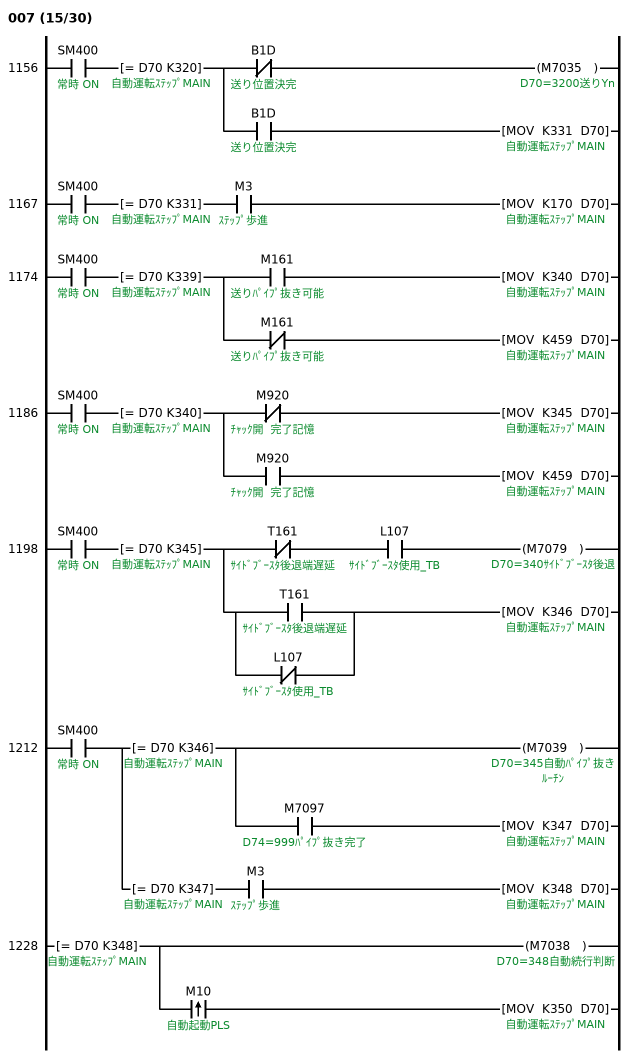
1156  LD      SM400  ; 常時 ON
      AND=    D70 K320  ; 自動運転ｽﾃｯﾌﾟMAIN
      MPS
      ANI     B1D  ; 送り位置決完
      OUT     M7035  ; D70=3200送りYn
      MPP
      AND     B1D  ; 送り位置決完
      MOV     K331 D70
1167  LD      SM400  ; 常時 ON
      AND=    D70 K331  ; 自動運転ｽﾃｯﾌﾟMAIN
      AND     M3  ; ｽﾃｯﾌﾟ歩進
      MOV     K170 D70
1174  LD      SM400  ; 常時 ON
      AND=    D70 K339  ; 自動運転ｽﾃｯﾌﾟMAIN
      MPS
      AND     M161  ; 送りﾊﾟｲﾌﾟ抜き可能
      MOV     K340 D70
      MPP
      ANI     M161  ; 送りﾊﾟｲﾌﾟ抜き可能
      MOV     K459 D70
1186  LD      SM400  ; 常時 ON
      AND=    D70 K340  ; 自動運転ｽﾃｯﾌﾟMAIN
      MPS
      ANI     M920  ; ﾁｬｯｸ開  完了記憶
      MOV     K345 D70
      MPP
      AND     M920  ; ﾁｬｯｸ開  完了記憶
      MOV     K459 D70
1198  LD      SM400  ; 常時 ON
      AND=    D70 K345  ; 自動運転ｽﾃｯﾌﾟMAIN
      MPS
      ANI     T161  ; ｻｲﾄﾞﾌﾞｰｽﾀ後退端遅延
      AND     L107  ; ｻｲﾄﾞﾌﾞｰｽﾀ使用_TB
      OUT     M7079  ; D70=340ｻｲﾄﾞﾌﾞｰｽﾀ後退
      MPP
      LD      T161  ; ｻｲﾄﾞﾌﾞｰｽﾀ後退端遅延
      ORI     L107  ; ｻｲﾄﾞﾌﾞｰｽﾀ使用_TB
      ANB
      MOV     K346 D70
1212  LD      SM400  ; 常時 ON
      MPS
      AND=    D70 K346  ; 自動運転ｽﾃｯﾌﾟMAIN
      OUT     M7039  ; D70=345自動ﾊﾟｲﾌﾟ抜きﾙｰﾁﾝ
      AND     M7097  ; D74=999ﾊﾟｲﾌﾟ抜き完了
      MOV     K347 D70
      MPP
      AND=    D70 K347  ; 自動運転ｽﾃｯﾌﾟMAIN
      AND     M3  ; ｽﾃｯﾌﾟ歩進
      MOV     K348 D70
1228  LD=     D70 K348  ; 自動運転ｽﾃｯﾌﾟMAIN
      OUT     M7038  ; D70=348自動続行判断
      ANDP    M10  ; 自動起動PLS
      MOV     K350 D70
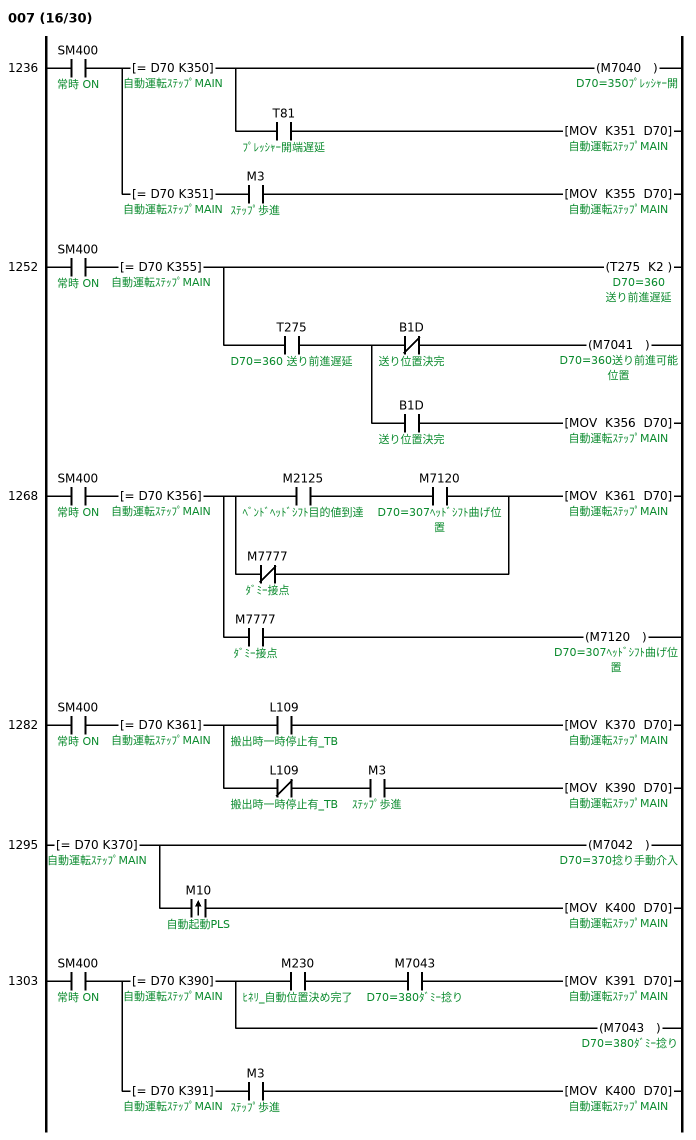
1236  LD      SM400  ; 常時 ON
      MPS
      AND=    D70 K350  ; 自動運転ｽﾃｯﾌﾟMAIN
      OUT     M7040  ; D70=350ﾌﾟﾚｯｼｬｰ開
      AND     T81  ; ﾌﾟﾚｯｼｬｰ開端遅延
      MOV     K351 D70
      MPP
      AND=    D70 K351  ; 自動運転ｽﾃｯﾌﾟMAIN
      AND     M3  ; ｽﾃｯﾌﾟ歩進
      MOV     K355 D70
1252  LD      SM400  ; 常時 ON
      AND=    D70 K355  ; 自動運転ｽﾃｯﾌﾟMAIN
      OUT     T275 K2  ; D70=360 送り前進遅延
      AND     T275  ; D70=360 送り前進遅延
      MPS
      ANI     B1D  ; 送り位置決完
      OUT     M7041  ; D70=360送り前進可能位置
      MPP
      AND     B1D  ; 送り位置決完
      MOV     K356 D70
1268  LD      SM400  ; 常時 ON
      AND=    D70 K356  ; 自動運転ｽﾃｯﾌﾟMAIN
      MPS
      LD      M2125  ; ﾍﾞﾝﾄﾞﾍｯﾄﾞｼﾌﾄ目的値到達
      AND     M7120  ; D70=307ﾍｯﾄﾞｼﾌﾄ曲げ位置
      ORI     M7777  ; ﾀﾞﾐｰ接点
      ANB
      MOV     K361 D70
      MPP
      AND     M7777  ; ﾀﾞﾐｰ接点
      OUT     M7120  ; D70=307ﾍｯﾄﾞｼﾌﾄ曲げ位置
1282  LD      SM400  ; 常時 ON
      AND=    D70 K361  ; 自動運転ｽﾃｯﾌﾟMAIN
      MPS
      AND     L109  ; 搬出時一時停止有_TB
      MOV     K370 D70
      MPP
      ANI     L109  ; 搬出時一時停止有_TB
      AND     M3  ; ｽﾃｯﾌﾟ歩進
      MOV     K390 D70
1295  LD=     D70 K370  ; 自動運転ｽﾃｯﾌﾟMAIN
      OUT     M7042  ; D70=370捻り手動介入
      ANDP    M10  ; 自動起動PLS
      MOV     K400 D70
1303  LD      SM400  ; 常時 ON
      MPS
      AND=    D70 K390  ; 自動運転ｽﾃｯﾌﾟMAIN
      MPS
      AND     M230  ; ﾋﾈﾘ_自動位置決め完了
      AND     M7043  ; D70=380ﾀﾞﾐｰ捻り
      MOV     K391 D70
      MPP
      OUT     M7043  ; D70=380ﾀﾞﾐｰ捻り
      MPP
      AND=    D70 K391  ; 自動運転ｽﾃｯﾌﾟMAIN
      AND     M3  ; ｽﾃｯﾌﾟ歩進
      MOV     K400 D70
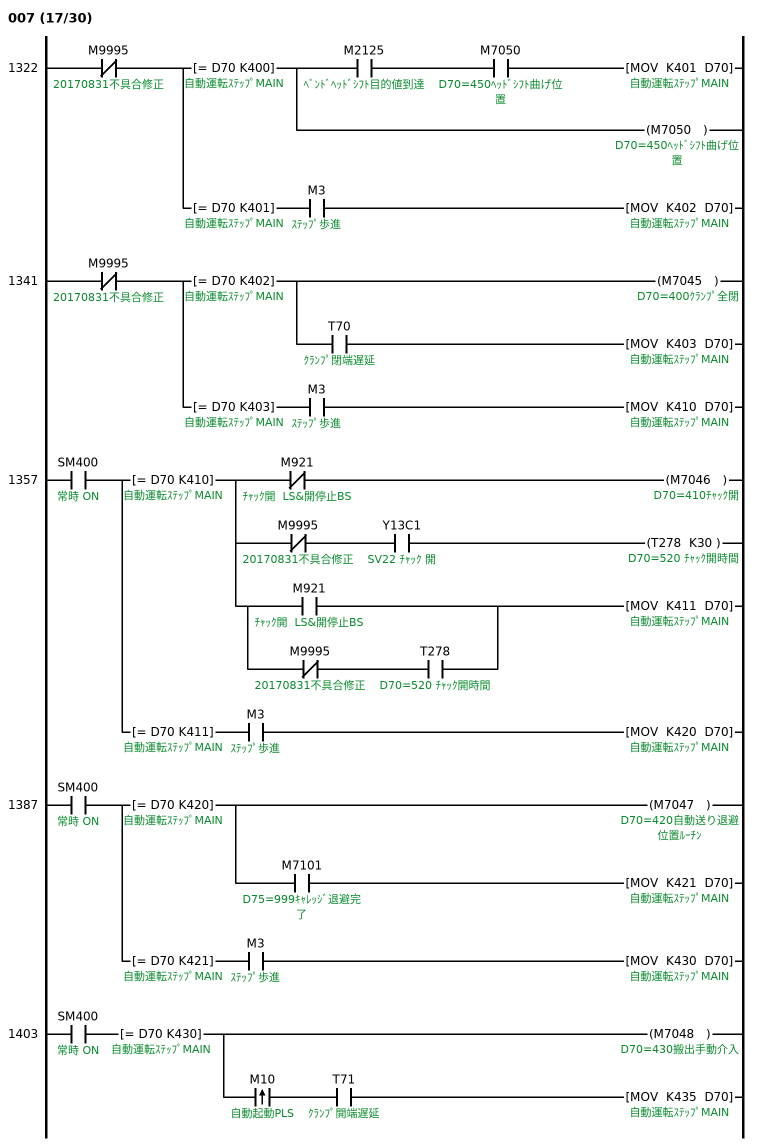
1322  LDI     M9995  ; 20170831不具合修正
      MPS
      AND=    D70 K400  ; 自動運転ｽﾃｯﾌﾟMAIN
      MPS
      AND     M2125  ; ﾍﾞﾝﾄﾞﾍｯﾄﾞｼﾌﾄ目的値到達
      AND     M7050  ; D70=450ﾍｯﾄﾞｼﾌﾄ曲げ位置
      MOV     K401 D70
      MPP
      OUT     M7050  ; D70=450ﾍｯﾄﾞｼﾌﾄ曲げ位置
      MPP
      AND=    D70 K401  ; 自動運転ｽﾃｯﾌﾟMAIN
      AND     M3  ; ｽﾃｯﾌﾟ歩進
      MOV     K402 D70
1341  LDI     M9995  ; 20170831不具合修正
      MPS
      AND=    D70 K402  ; 自動運転ｽﾃｯﾌﾟMAIN
      OUT     M7045  ; D70=400ｸﾗﾝﾌﾟ全閉
      AND     T70  ; ｸﾗﾝﾌﾟ閉端遅延
      MOV     K403 D70
      MPP
      AND=    D70 K403  ; 自動運転ｽﾃｯﾌﾟMAIN
      AND     M3  ; ｽﾃｯﾌﾟ歩進
      MOV     K410 D70
1357  LD      SM400  ; 常時 ON
      MPS
      AND=    D70 K410  ; 自動運転ｽﾃｯﾌﾟMAIN
      MPS
      ANI     M921  ; ﾁｬｯｸ開  LS&開停止BS
      OUT     M7046  ; D70=410ﾁｬｯｸ開
      MRD
      ANI     M9995  ; 20170831不具合修正
      AND     Y13C1  ; SV22 ﾁｬｯｸ 開
      OUT     T278 K30  ; D70=520 ﾁｬｯｸ開時間
      MPP
      LD      M921  ; ﾁｬｯｸ開  LS&開停止BS
      LDI     M9995  ; 20170831不具合修正
      AND     T278  ; D70=520 ﾁｬｯｸ開時間
      ORB
      ANB
      MOV     K411 D70
      MPP
      AND=    D70 K411  ; 自動運転ｽﾃｯﾌﾟMAIN
      AND     M3  ; ｽﾃｯﾌﾟ歩進
      MOV     K420 D70
1387  LD      SM400  ; 常時 ON
      MPS
      AND=    D70 K420  ; 自動運転ｽﾃｯﾌﾟMAIN
      OUT     M7047  ; D70=420自動送り退避位置ﾙｰﾁﾝ
      AND     M7101  ; D75=999ｷｬﾚｯｼﾞ退避完了
      MOV     K421 D70
      MPP
      AND=    D70 K421  ; 自動運転ｽﾃｯﾌﾟMAIN
      AND     M3  ; ｽﾃｯﾌﾟ歩進
      MOV     K430 D70
1403  LD      SM400  ; 常時 ON
      AND=    D70 K430  ; 自動運転ｽﾃｯﾌﾟMAIN
      OUT     M7048  ; D70=430搬出手動介入
      ANDP    M10  ; 自動起動PLS
      AND     T71  ; ｸﾗﾝﾌﾟ開端遅延
      MOV     K435 D70
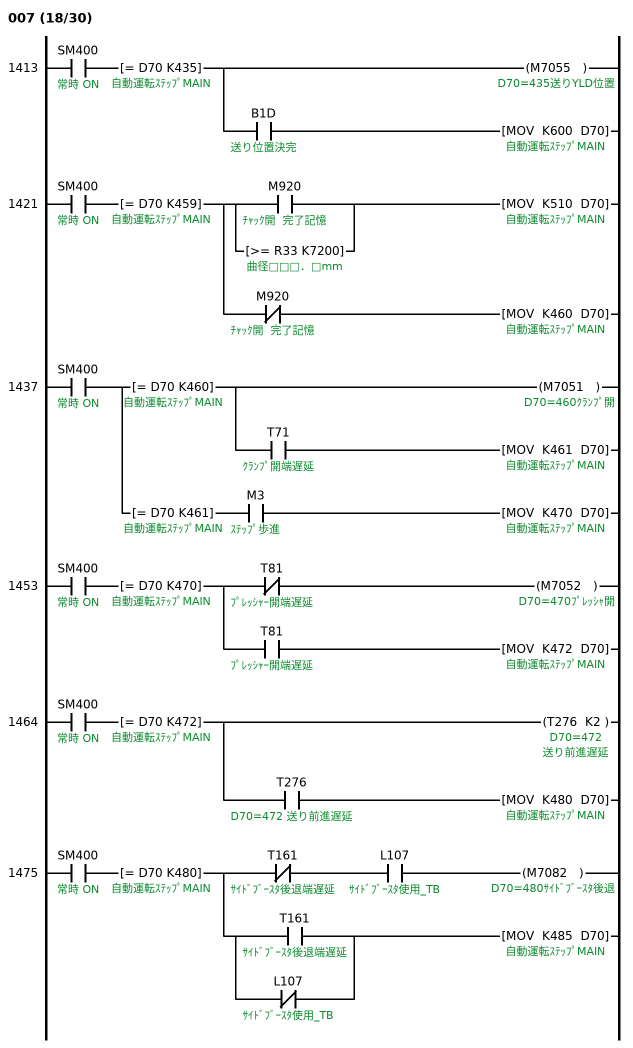
1413  LD      SM400  ; 常時 ON
      AND=    D70 K435  ; 自動運転ｽﾃｯﾌﾟMAIN
      OUT     M7055  ; D70=435送りYLD位置
      AND     B1D  ; 送り位置決完
      MOV     K600 D70
1421  LD      SM400  ; 常時 ON
      AND=    D70 K459  ; 自動運転ｽﾃｯﾌﾟMAIN
      MPS
      LD      M920  ; ﾁｬｯｸ開  完了記憶
      OR>=    R33 K7200  ; 曲径□□□．□mm
      ANB
      MOV     K510 D70
      MPP
      ANI     M920  ; ﾁｬｯｸ開  完了記憶
      MOV     K460 D70
1437  LD      SM400  ; 常時 ON
      MPS
      AND=    D70 K460  ; 自動運転ｽﾃｯﾌﾟMAIN
      OUT     M7051  ; D70=460ｸﾗﾝﾌﾟ開
      AND     T71  ; ｸﾗﾝﾌﾟ開端遅延
      MOV     K461 D70
      MPP
      AND=    D70 K461  ; 自動運転ｽﾃｯﾌﾟMAIN
      AND     M3  ; ｽﾃｯﾌﾟ歩進
      MOV     K470 D70
1453  LD      SM400  ; 常時 ON
      AND=    D70 K470  ; 自動運転ｽﾃｯﾌﾟMAIN
      MPS
      ANI     T81  ; ﾌﾟﾚｯｼｬｰ開端遅延
      OUT     M7052  ; D70=470ﾌﾟﾚｯｼｬ開
      MPP
      AND     T81  ; ﾌﾟﾚｯｼｬｰ開端遅延
      MOV     K472 D70
1464  LD      SM400  ; 常時 ON
      AND=    D70 K472  ; 自動運転ｽﾃｯﾌﾟMAIN
      OUT     T276 K2  ; D70=472 送り前進遅延
      AND     T276  ; D70=472 送り前進遅延
      MOV     K480 D70
1475  LD      SM400  ; 常時 ON
      AND=    D70 K480  ; 自動運転ｽﾃｯﾌﾟMAIN
      MPS
      ANI     T161  ; ｻｲﾄﾞﾌﾞｰｽﾀ後退端遅延
      AND     L107  ; ｻｲﾄﾞﾌﾞｰｽﾀ使用_TB
      OUT     M7082  ; D70=480ｻｲﾄﾞﾌﾞｰｽﾀ後退
      MPP
      LD      T161  ; ｻｲﾄﾞﾌﾞｰｽﾀ後退端遅延
      ORI     L107  ; ｻｲﾄﾞﾌﾞｰｽﾀ使用_TB
      ANB
      MOV     K485 D70
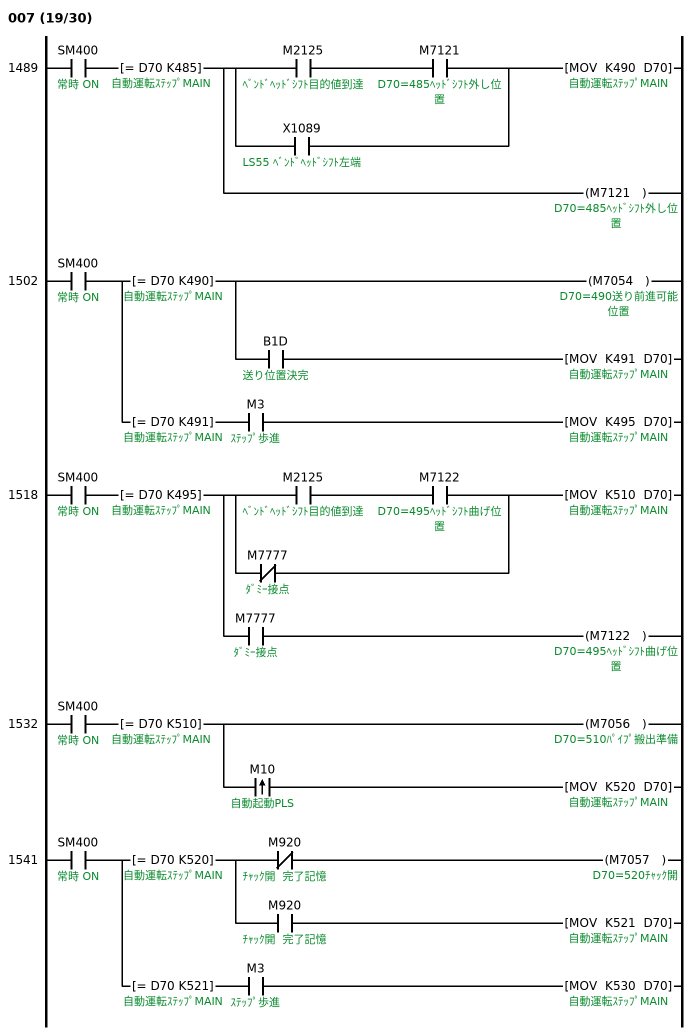
1489  LD      SM400  ; 常時 ON
      AND=    D70 K485  ; 自動運転ｽﾃｯﾌﾟMAIN
      MPS
      LD      M2125  ; ﾍﾞﾝﾄﾞﾍｯﾄﾞｼﾌﾄ目的値到達
      AND     M7121  ; D70=485ﾍｯﾄﾞｼﾌﾄ外し位置
      OR      X1089  ; LS55 ﾍﾞﾝﾄﾞﾍｯﾄﾞｼﾌﾄ左端
      ANB
      MOV     K490 D70
      MPP
      OUT     M7121  ; D70=485ﾍｯﾄﾞｼﾌﾄ外し位置
1502  LD      SM400  ; 常時 ON
      MPS
      AND=    D70 K490  ; 自動運転ｽﾃｯﾌﾟMAIN
      OUT     M7054  ; D70=490送り前進可能位置
      AND     B1D  ; 送り位置決完
      MOV     K491 D70
      MPP
      AND=    D70 K491  ; 自動運転ｽﾃｯﾌﾟMAIN
      AND     M3  ; ｽﾃｯﾌﾟ歩進
      MOV     K495 D70
1518  LD      SM400  ; 常時 ON
      AND=    D70 K495  ; 自動運転ｽﾃｯﾌﾟMAIN
      MPS
      LD      M2125  ; ﾍﾞﾝﾄﾞﾍｯﾄﾞｼﾌﾄ目的値到達
      AND     M7122  ; D70=495ﾍｯﾄﾞｼﾌﾄ曲げ位置
      ORI     M7777  ; ﾀﾞﾐｰ接点
      ANB
      MOV     K510 D70
      MPP
      AND     M7777  ; ﾀﾞﾐｰ接点
      OUT     M7122  ; D70=495ﾍｯﾄﾞｼﾌﾄ曲げ位置
1532  LD      SM400  ; 常時 ON
      AND=    D70 K510  ; 自動運転ｽﾃｯﾌﾟMAIN
      OUT     M7056  ; D70=510ﾊﾟｲﾌﾟ搬出準備
      ANDP    M10  ; 自動起動PLS
      MOV     K520 D70
1541  LD      SM400  ; 常時 ON
      MPS
      AND=    D70 K520  ; 自動運転ｽﾃｯﾌﾟMAIN
      MPS
      ANI     M920  ; ﾁｬｯｸ開  完了記憶
      OUT     M7057  ; D70=520ﾁｬｯｸ開
      MPP
      AND     M920  ; ﾁｬｯｸ開  完了記憶
      MOV     K521 D70
      MPP
      AND=    D70 K521  ; 自動運転ｽﾃｯﾌﾟMAIN
      AND     M3  ; ｽﾃｯﾌﾟ歩進
      MOV     K530 D70
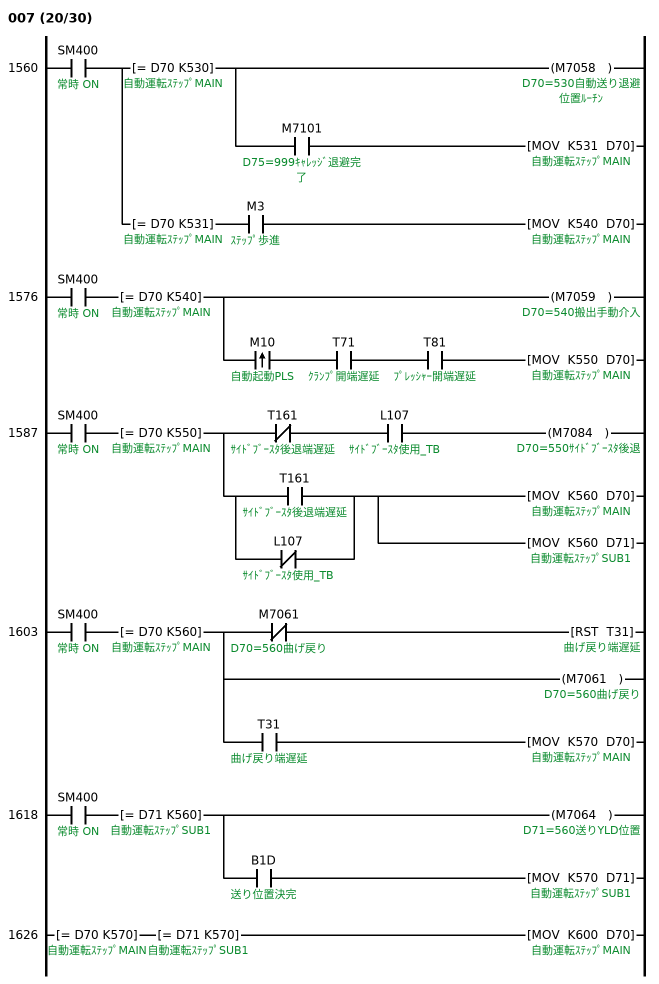
1560  LD      SM400  ; 常時 ON
      MPS
      AND=    D70 K530  ; 自動運転ｽﾃｯﾌﾟMAIN
      OUT     M7058  ; D70=530自動送り退避位置ﾙｰﾁﾝ
      AND     M7101  ; D75=999ｷｬﾚｯｼﾞ退避完了
      MOV     K531 D70
      MPP
      AND=    D70 K531  ; 自動運転ｽﾃｯﾌﾟMAIN
      AND     M3  ; ｽﾃｯﾌﾟ歩進
      MOV     K540 D70
1576  LD      SM400  ; 常時 ON
      AND=    D70 K540  ; 自動運転ｽﾃｯﾌﾟMAIN
      OUT     M7059  ; D70=540搬出手動介入
      ANDP    M10  ; 自動起動PLS
      AND     T71  ; ｸﾗﾝﾌﾟ開端遅延
      AND     T81  ; ﾌﾟﾚｯｼｬｰ開端遅延
      MOV     K550 D70
1587  LD      SM400  ; 常時 ON
      AND=    D70 K550  ; 自動運転ｽﾃｯﾌﾟMAIN
      MPS
      ANI     T161  ; ｻｲﾄﾞﾌﾞｰｽﾀ後退端遅延
      AND     L107  ; ｻｲﾄﾞﾌﾞｰｽﾀ使用_TB
      OUT     M7084  ; D70=550ｻｲﾄﾞﾌﾞｰｽﾀ後退
      MPP
      LD      T161  ; ｻｲﾄﾞﾌﾞｰｽﾀ後退端遅延
      ORI     L107  ; ｻｲﾄﾞﾌﾞｰｽﾀ使用_TB
      ANB
      MOV     K560 D70
      MOV     K560 D71
1603  LD      SM400  ; 常時 ON
      AND=    D70 K560  ; 自動運転ｽﾃｯﾌﾟMAIN
      MPS
      ANI     M7061  ; D70=560曲げ戻り
      RST     T31  ; 曲げ戻り端遅延
      MPP
      OUT     M7061  ; D70=560曲げ戻り
      AND     T31  ; 曲げ戻り端遅延
      MOV     K570 D70
1618  LD      SM400  ; 常時 ON
      AND=    D71 K560  ; 自動運転ｽﾃｯﾌﾟSUB1
      OUT     M7064  ; D71=560送りYLD位置
      AND     B1D  ; 送り位置決完
      MOV     K570 D71
1626  LD=     D70 K570  ; 自動運転ｽﾃｯﾌﾟMAIN
      AND=    D71 K570  ; 自動運転ｽﾃｯﾌﾟSUB1
      MOV     K600 D70
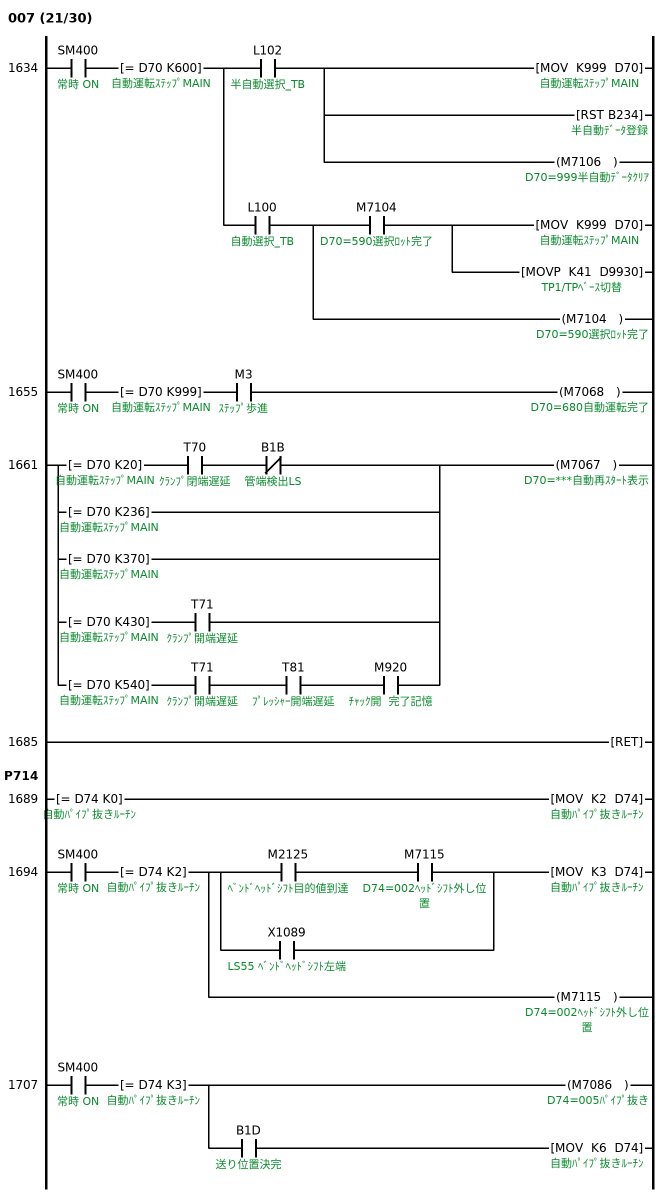
1634  LD      SM400  ; 常時 ON
      AND=    D70 K600  ; 自動運転ｽﾃｯﾌﾟMAIN
      MPS
      AND     L102  ; 半自動選択_TB
      MOV     K999 D70
      RST     B234  ; 半自動ﾃﾞｰﾀ登録
      OUT     M7106  ; D70=999半自動ﾃﾞｰﾀｸﾘｱ
      MPP
      AND     L100  ; 自動選択_TB
      MPS
      AND     M7104  ; D70=590選択ﾛｯﾄ完了
      MOV     K999 D70
      MOVP    K41 D9930  ; TP1/TPﾍﾞｰｽ切替
      MPP
      OUT     M7104  ; D70=590選択ﾛｯﾄ完了
1655  LD      SM400  ; 常時 ON
      AND=    D70 K999  ; 自動運転ｽﾃｯﾌﾟMAIN
      AND     M3  ; ｽﾃｯﾌﾟ歩進
      OUT     M7068  ; D70=680自動運転完了
1661  LD=     D70 K20  ; 自動運転ｽﾃｯﾌﾟMAIN
      AND     T70  ; ｸﾗﾝﾌﾟ閉端遅延
      ANI     B1B  ; 管端検出LS
      OR=     D70 K236  ; 自動運転ｽﾃｯﾌﾟMAIN
      OR=     D70 K370  ; 自動運転ｽﾃｯﾌﾟMAIN
      LD=     D70 K430  ; 自動運転ｽﾃｯﾌﾟMAIN
      AND     T71  ; ｸﾗﾝﾌﾟ開端遅延
      ORB
      LD=     D70 K540  ; 自動運転ｽﾃｯﾌﾟMAIN
      AND     T71  ; ｸﾗﾝﾌﾟ開端遅延
      AND     T81  ; ﾌﾟﾚｯｼｬｰ開端遅延
      AND     M920  ; ﾁｬｯｸ開  完了記憶
      ORB
      OUT     M7067  ; D70=***自動再ｽﾀｰﾄ表示
1685  RET
; 
      P714
1689  LD=     D74 K0  ; 自動ﾊﾟｲﾌﾟ抜きﾙｰﾁﾝ
      MOV     K2 D74
1694  LD      SM400  ; 常時 ON
      AND=    D74 K2  ; 自動ﾊﾟｲﾌﾟ抜きﾙｰﾁﾝ
      MPS
      LD      M2125  ; ﾍﾞﾝﾄﾞﾍｯﾄﾞｼﾌﾄ目的値到達
      AND     M7115  ; D74=002ﾍｯﾄﾞｼﾌﾄ外し位置
      OR      X1089  ; LS55 ﾍﾞﾝﾄﾞﾍｯﾄﾞｼﾌﾄ左端
      ANB
      MOV     K3 D74
      MPP
      OUT     M7115  ; D74=002ﾍｯﾄﾞｼﾌﾄ外し位置
1707  LD      SM400  ; 常時 ON
      AND=    D74 K3  ; 自動ﾊﾟｲﾌﾟ抜きﾙｰﾁﾝ
      OUT     M7086  ; D74=005ﾊﾟｲﾌﾟ抜き
      AND     B1D  ; 送り位置決完
      MOV     K6 D74
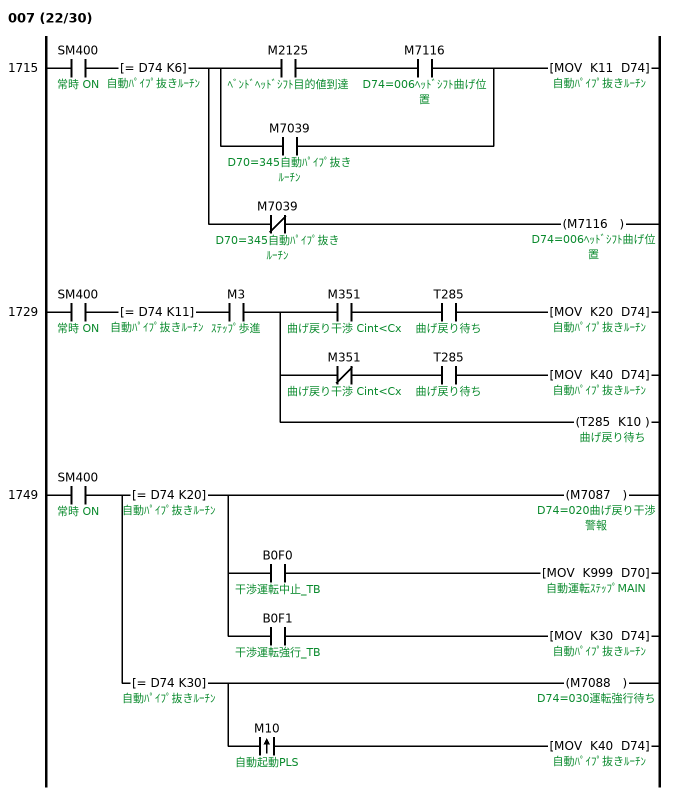
1715  LD      SM400  ; 常時 ON
      AND=    D74 K6  ; 自動ﾊﾟｲﾌﾟ抜きﾙｰﾁﾝ
      MPS
      LD      M2125  ; ﾍﾞﾝﾄﾞﾍｯﾄﾞｼﾌﾄ目的値到達
      AND     M7116  ; D74=006ﾍｯﾄﾞｼﾌﾄ曲げ位置
      OR      M7039  ; D70=345自動ﾊﾟｲﾌﾟ抜きﾙｰﾁﾝ
      ANB
      MOV     K11 D74
      MPP
      ANI     M7039  ; D70=345自動ﾊﾟｲﾌﾟ抜きﾙｰﾁﾝ
      OUT     M7116  ; D74=006ﾍｯﾄﾞｼﾌﾄ曲げ位置
1729  LD      SM400  ; 常時 ON
      AND=    D74 K11  ; 自動ﾊﾟｲﾌﾟ抜きﾙｰﾁﾝ
      AND     M3  ; ｽﾃｯﾌﾟ歩進
      MPS
      AND     M351  ; 曲げ戻り干渉 Cint<Cx
      AND     T285  ; 曲げ戻り待ち
      MOV     K20 D74
      MRD
      ANI     M351  ; 曲げ戻り干渉 Cint<Cx
      AND     T285  ; 曲げ戻り待ち
      MOV     K40 D74
      MPP
      OUT     T285 K10  ; 曲げ戻り待ち
1749  LD      SM400  ; 常時 ON
      MPS
      AND=    D74 K20  ; 自動ﾊﾟｲﾌﾟ抜きﾙｰﾁﾝ
      OUT     M7087  ; D74=020曲げ戻り干渉警報
      MPS
      AND     B0F0  ; 干渉運転中止_TB
      MOV     K999 D70
      MPP
      AND     B0F1  ; 干渉運転強行_TB
      MOV     K30 D74
      MPP
      AND=    D74 K30  ; 自動ﾊﾟｲﾌﾟ抜きﾙｰﾁﾝ
      OUT     M7088  ; D74=030運転強行待ち
      ANDP    M10  ; 自動起動PLS
      MOV     K40 D74
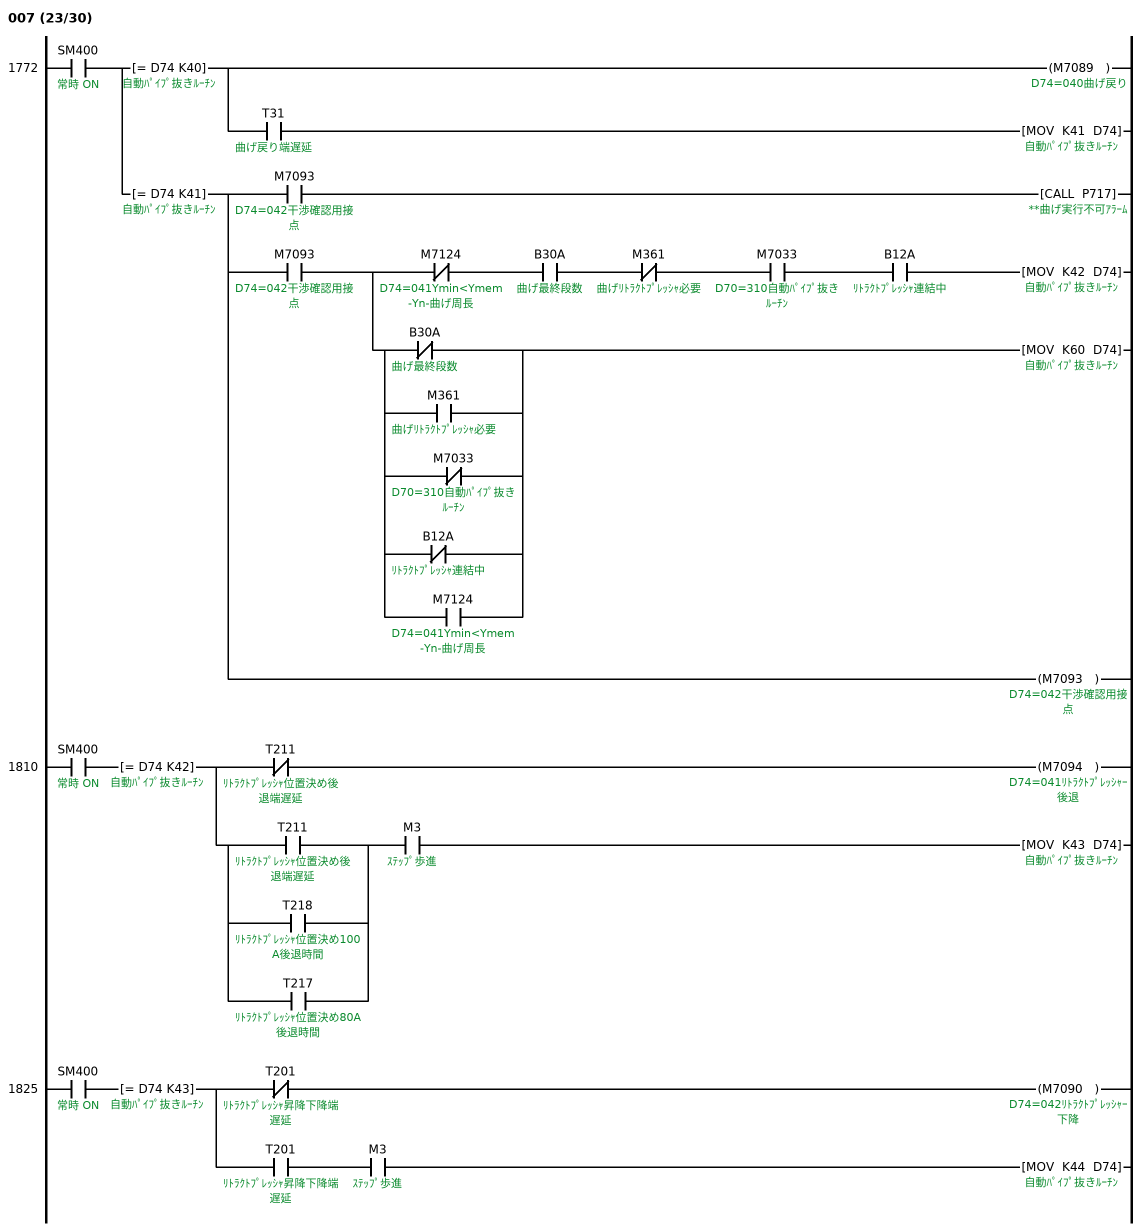
1772  LD      SM400  ; 常時 ON
      MPS
      AND=    D74 K40  ; 自動ﾊﾟｲﾌﾟ抜きﾙｰﾁﾝ
      OUT     M7089  ; D74=040曲げ戻り
      AND     T31  ; 曲げ戻り端遅延
      MOV     K41 D74
      MPP
      AND=    D74 K41  ; 自動ﾊﾟｲﾌﾟ抜きﾙｰﾁﾝ
      MPS
      AND     M7093  ; D74=042干渉確認用接点
      CALL    P717
      MRD
      AND     M7093  ; D74=042干渉確認用接点
      MPS
      ANI     M7124  ; D74=041Ymin<Ymem-Yn-曲げ周長
      AND     B30A  ; 曲げ最終段数
      ANI     M361  ; 曲げﾘﾄﾗｸﾄﾌﾟﾚｯｼｬ必要
      AND     M7033  ; D70=310自動ﾊﾟｲﾌﾟ抜きﾙｰﾁﾝ
      AND     B12A  ; ﾘﾄﾗｸﾄﾌﾟﾚｯｼｬ連結中
      MOV     K42 D74
      MPP
      LDI     B30A  ; 曲げ最終段数
      OR      M361  ; 曲げﾘﾄﾗｸﾄﾌﾟﾚｯｼｬ必要
      ORI     M7033  ; D70=310自動ﾊﾟｲﾌﾟ抜きﾙｰﾁﾝ
      ORI     B12A  ; ﾘﾄﾗｸﾄﾌﾟﾚｯｼｬ連結中
      OR      M7124  ; D74=041Ymin<Ymem-Yn-曲げ周長
      ANB
      MOV     K60 D74
      MPP
      OUT     M7093  ; D74=042干渉確認用接点
1810  LD      SM400  ; 常時 ON
      AND=    D74 K42  ; 自動ﾊﾟｲﾌﾟ抜きﾙｰﾁﾝ
      MPS
      ANI     T211  ; ﾘﾄﾗｸﾄﾌﾟﾚｯｼｬ位置決め後退端遅延
      OUT     M7094  ; D74=041ﾘﾄﾗｸﾄﾌﾟﾚｯｼｬｰ後退
      MPP
      LD      T211  ; ﾘﾄﾗｸﾄﾌﾟﾚｯｼｬ位置決め後退端遅延
      OR      T218  ; ﾘﾄﾗｸﾄﾌﾟﾚｯｼｬ位置決め100A後退時間
      OR      T217  ; ﾘﾄﾗｸﾄﾌﾟﾚｯｼｬ位置決め80A後退時間
      ANB
      AND     M3  ; ｽﾃｯﾌﾟ歩進
      MOV     K43 D74
1825  LD      SM400  ; 常時 ON
      AND=    D74 K43  ; 自動ﾊﾟｲﾌﾟ抜きﾙｰﾁﾝ
      MPS
      ANI     T201  ; ﾘﾄﾗｸﾄﾌﾟﾚｯｼｬ昇降下降端遅延
      OUT     M7090  ; D74=042ﾘﾄﾗｸﾄﾌﾟﾚｯｼｬｰ下降
      MPP
      AND     T201  ; ﾘﾄﾗｸﾄﾌﾟﾚｯｼｬ昇降下降端遅延
      AND     M3  ; ｽﾃｯﾌﾟ歩進
      MOV     K44 D74
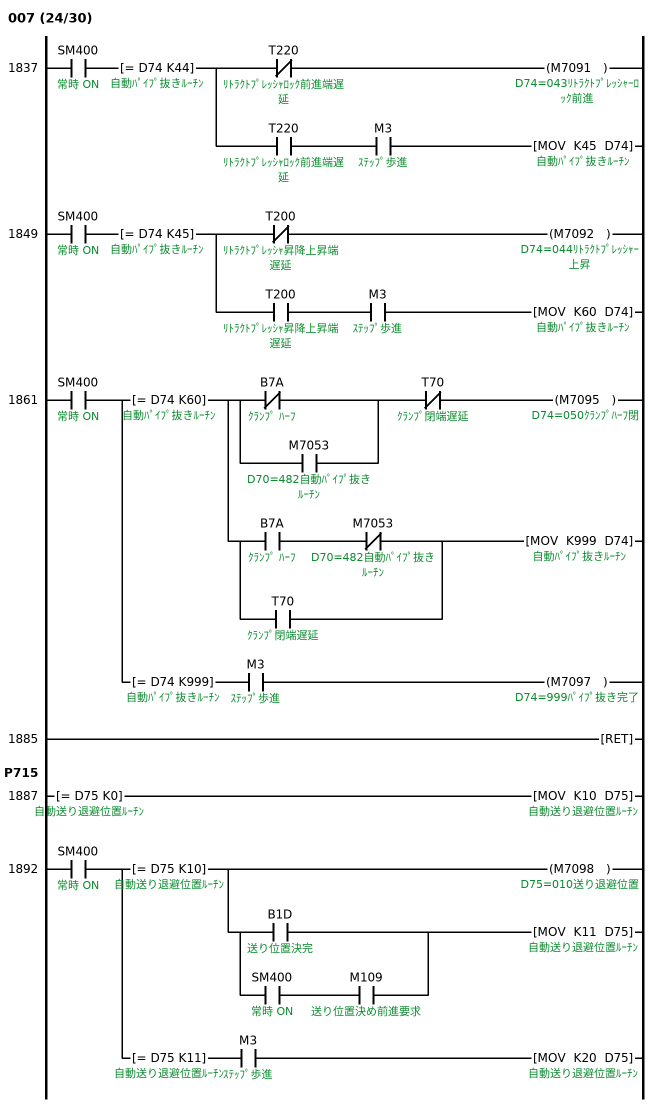
1837  LD      SM400  ; 常時 ON
      AND=    D74 K44  ; 自動ﾊﾟｲﾌﾟ抜きﾙｰﾁﾝ
      MPS
      ANI     T220  ; ﾘﾄﾗｸﾄﾌﾟﾚｯｼｬﾛｯｸ前進端遅延
      OUT     M7091  ; D74=043ﾘﾄﾗｸﾄﾌﾟﾚｯｼｬｰﾛｯｸ前進
      MPP
      AND     T220  ; ﾘﾄﾗｸﾄﾌﾟﾚｯｼｬﾛｯｸ前進端遅延
      AND     M3  ; ｽﾃｯﾌﾟ歩進
      MOV     K45 D74
1849  LD      SM400  ; 常時 ON
      AND=    D74 K45  ; 自動ﾊﾟｲﾌﾟ抜きﾙｰﾁﾝ
      MPS
      ANI     T200  ; ﾘﾄﾗｸﾄﾌﾟﾚｯｼｬ昇降上昇端遅延
      OUT     M7092  ; D74=044ﾘﾄﾗｸﾄﾌﾟﾚｯｼｬｰ上昇
      MPP
      AND     T200  ; ﾘﾄﾗｸﾄﾌﾟﾚｯｼｬ昇降上昇端遅延
      AND     M3  ; ｽﾃｯﾌﾟ歩進
      MOV     K60 D74
1861  LD      SM400  ; 常時 ON
      MPS
      AND=    D74 K60  ; 自動ﾊﾟｲﾌﾟ抜きﾙｰﾁﾝ
      MPS
      LDI     B7A  ; ｸﾗﾝﾌﾟ ﾊｰﾌ
      OR      M7053  ; D70=482自動ﾊﾟｲﾌﾟ抜きﾙｰﾁﾝ
      ANB
      ANI     T70  ; ｸﾗﾝﾌﾟ閉端遅延
      OUT     M7095  ; D74=050ｸﾗﾝﾌﾟﾊｰﾌ閉
      MPP
      LD      B7A  ; ｸﾗﾝﾌﾟ ﾊｰﾌ
      ANI     M7053  ; D70=482自動ﾊﾟｲﾌﾟ抜きﾙｰﾁﾝ
      OR      T70  ; ｸﾗﾝﾌﾟ閉端遅延
      ANB
      MOV     K999 D74
      MPP
      AND=    D74 K999  ; 自動ﾊﾟｲﾌﾟ抜きﾙｰﾁﾝ
      AND     M3  ; ｽﾃｯﾌﾟ歩進
      OUT     M7097  ; D74=999ﾊﾟｲﾌﾟ抜き完了
1885  RET
      P715
1887  LD=     D75 K0  ; 自動送り退避位置ﾙｰﾁﾝ
      MOV     K10 D75
1892  LD      SM400  ; 常時 ON
      MPS
      AND=    D75 K10  ; 自動送り退避位置ﾙｰﾁﾝ
      OUT     M7098  ; D75=010送り退避位置
      LD      B1D  ; 送り位置決完
      LD      SM400  ; 常時 ON
      AND     M109  ; 送り位置決め前進要求
      ORB
      ANB
      MOV     K11 D75
      MPP
      AND=    D75 K11  ; 自動送り退避位置ﾙｰﾁﾝ
      AND     M3  ; ｽﾃｯﾌﾟ歩進
      MOV     K20 D75
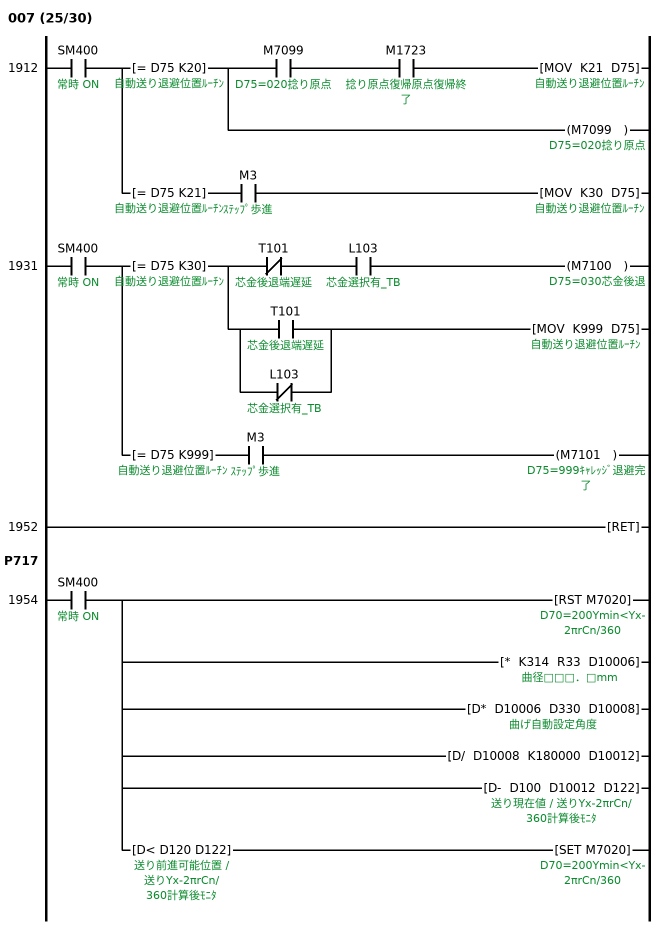
1912  LD      SM400  ; 常時 ON
      MPS
      AND=    D75 K20  ; 自動送り退避位置ﾙｰﾁﾝ
      MPS
      AND     M7099  ; D75=020捻り原点
      AND     M1723  ; 捻り原点復帰原点復帰終了
      MOV     K21 D75
      MPP
      OUT     M7099  ; D75=020捻り原点
      MPP
      AND=    D75 K21  ; 自動送り退避位置ﾙｰﾁﾝ
      AND     M3  ; ｽﾃｯﾌﾟ歩進
      MOV     K30 D75
1931  LD      SM400  ; 常時 ON
      MPS
      AND=    D75 K30  ; 自動送り退避位置ﾙｰﾁﾝ
      MPS
      ANI     T101  ; 芯金後退端遅延
      AND     L103  ; 芯金選択有_TB
      OUT     M7100  ; D75=030芯金後退
      MPP
      LD      T101  ; 芯金後退端遅延
      ORI     L103  ; 芯金選択有_TB
      ANB
      MOV     K999 D75
      MPP
      AND=    D75 K999  ; 自動送り退避位置ﾙｰﾁﾝ
      AND     M3  ; ｽﾃｯﾌﾟ歩進
      OUT     M7101  ; D75=999ｷｬﾚｯｼﾞ退避完了
1952  RET
      P717
1954  LD      SM400  ; 常時 ON
      RST     M7020  ; D70=200Ymin<Yx-2πrCn/360
      *       K314 R33 D10006
      D*      D10006 D330 D10008  ; 曲げ自動設定角度
      D/      D10008 K180000 D10012
      D-      D100 D10012 D122  ; 送りYx-2πrCn/360計算後ﾓﾆﾀ
      ANDD<   D120 D122  ; 送り前進可能位置 / 送りYx-2πrCn/360計算後ﾓﾆﾀ
      SET     M7020  ; D70=200Ymin<Yx-2πrCn/360
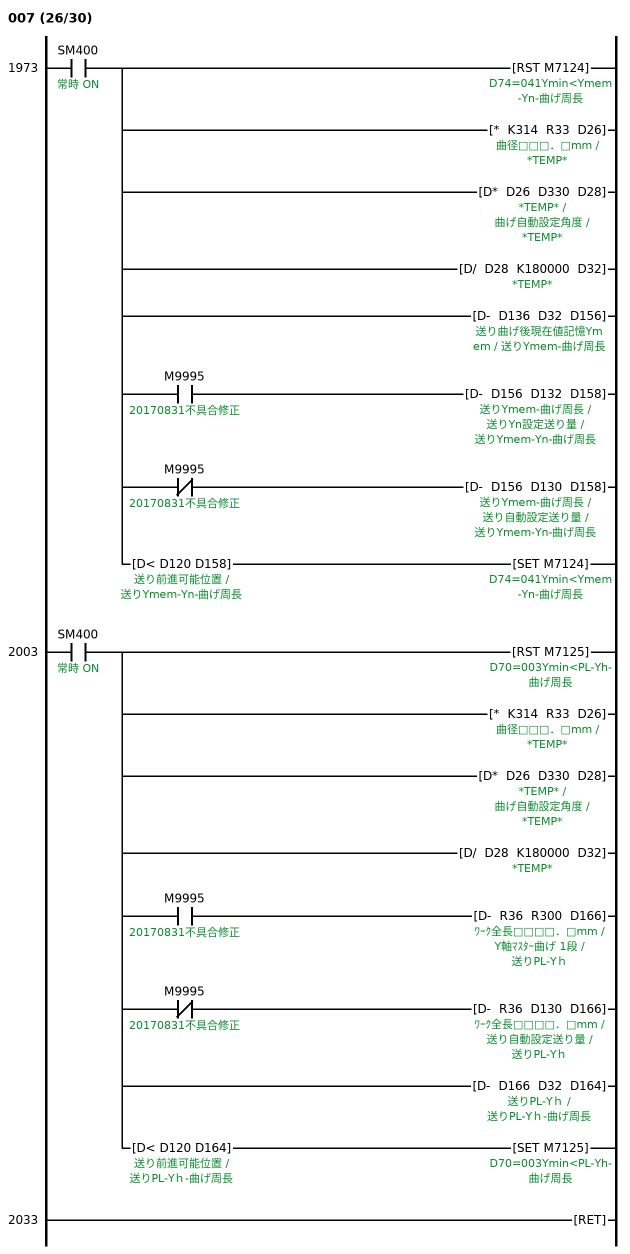
1973  LD      SM400  ; 常時 ON
      RST     M7124  ; D74=041Ymin<Ymem-Yn-曲げ周長
      *       K314 R33 D26  ; *TEMP*
      D*      D26 D330 D28  ; *TEMP*
      D/      D28 K180000 D32
      D-      D136 D32 D156  ; 送りYmem-曲げ周長
      MPS
      AND     M9995  ; 20170831不具合修正
      D-      D156 D132 D158  ; 送りYn設定送り量 / 送りYmem-Yn-曲げ周長
      MRD
      ANI     M9995  ; 20170831不具合修正
      D-      D156 D130 D158  ; 送り自動設定送り量
      MPP
      ANDD<   D120 D158  ; 送り前進可能位置 / 送りYmem-Yn-曲げ周長
      SET     M7124  ; D74=041Ymin<Ymem-Yn-曲げ周長
2003  LD      SM400  ; 常時 ON
      RST     M7125  ; D70=003Ymin<PL-Yh-曲げ周長
      *       K314 R33 D26
      D*      D26 D330 D28
      D/      D28 K180000 D32
      MPS
      AND     M9995  ; 20170831不具合修正
      D-      R36 R300 D166  ; ﾜｰｸ全長□□□□．□mm / Y軸ﾏｽﾀｰ曲げ 1段 / 送りPL-Yｈ
      MRD
      ANI     M9995  ; 20170831不具合修正
      D-      R36 D130 D166
      MPP
      D-      D166 D32 D164  ; 送りPL-Yｈ-曲げ周長
      ANDD<   D120 D164  ; 送り前進可能位置 / 送りPL-Yｈ-曲げ周長
      SET     M7125  ; D70=003Ymin<PL-Yh-曲げ周長
2033  RET
; 
      P720
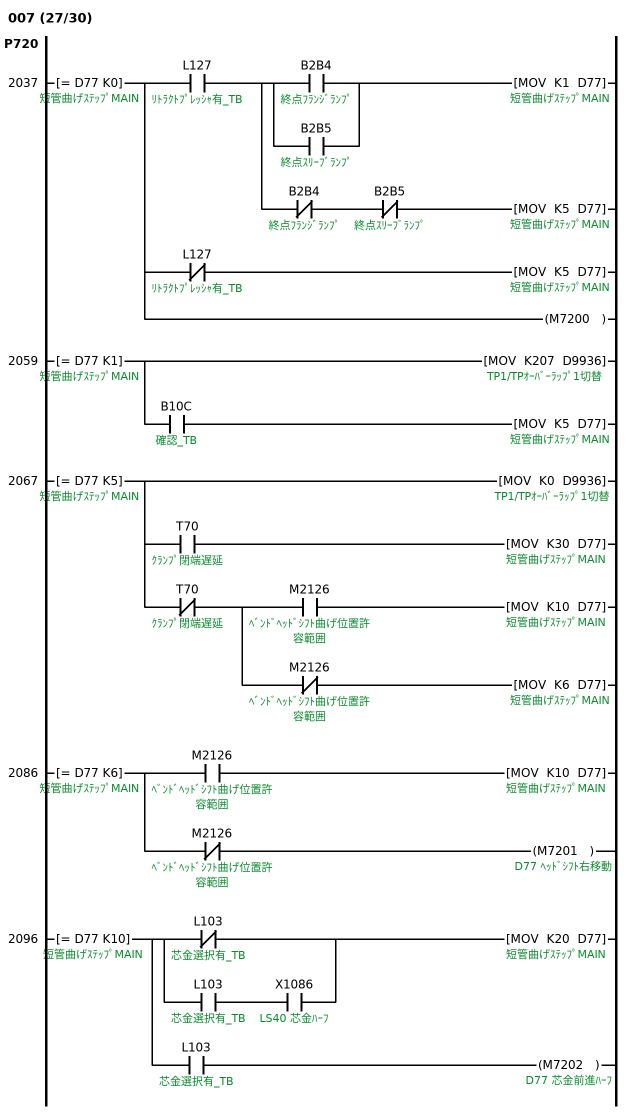
2037  LD=     D77 K0  ; 短管曲げｽﾃｯﾌﾟMAIN
      MPS
      AND     L127  ; ﾘﾄﾗｸﾄﾌﾟﾚｯｼｬ有_TB
      MPS
      LD      B2B4  ; 終点ﾌﾗﾝｼﾞﾗﾝﾌﾟ
      OR      B2B5  ; 終点ｽﾘｰﾌﾞﾗﾝﾌﾟ
      ANB
      MOV     K1 D77
      MPP
      ANI     B2B4  ; 終点ﾌﾗﾝｼﾞﾗﾝﾌﾟ
      ANI     B2B5  ; 終点ｽﾘｰﾌﾞﾗﾝﾌﾟ
      MOV     K5 D77
      MRD
      ANI     L127  ; ﾘﾄﾗｸﾄﾌﾟﾚｯｼｬ有_TB
      MOV     K5 D77
      MPP
      OUT     M7200
2059  LD=     D77 K1  ; 短管曲げｽﾃｯﾌﾟMAIN
      MOV     K207 D9936
      AND     B10C  ; 確認_TB
      MOV     K5 D77
2067  LD=     D77 K5  ; 短管曲げｽﾃｯﾌﾟMAIN
      MOV     K0 D9936
      MPS
      AND     T70  ; ｸﾗﾝﾌﾟ閉端遅延
      MOV     K30 D77
      MPP
      ANI     T70  ; ｸﾗﾝﾌﾟ閉端遅延
      MPS
      AND     M2126  ; ﾍﾞﾝﾄﾞﾍｯﾄﾞｼﾌﾄ曲げ位置許容範囲
      MOV     K10 D77
      MPP
      ANI     M2126  ; ﾍﾞﾝﾄﾞﾍｯﾄﾞｼﾌﾄ曲げ位置許容範囲
      MOV     K6 D77
2086  LD=     D77 K6  ; 短管曲げｽﾃｯﾌﾟMAIN
      MPS
      AND     M2126  ; ﾍﾞﾝﾄﾞﾍｯﾄﾞｼﾌﾄ曲げ位置許容範囲
      MOV     K10 D77
      MPP
      ANI     M2126  ; ﾍﾞﾝﾄﾞﾍｯﾄﾞｼﾌﾄ曲げ位置許容範囲
      OUT     M7201  ; D77 ﾍｯﾄﾞｼﾌﾄ右移動
2096  LD=     D77 K10  ; 短管曲げｽﾃｯﾌﾟMAIN
      MPS
      LDI     L103  ; 芯金選択有_TB
      LD      L103  ; 芯金選択有_TB
      AND     X1086  ; LS40 芯金ﾊｰﾌ
      ORB
      ANB
      MOV     K20 D77
      MPP
      AND     L103  ; 芯金選択有_TB
      OUT     M7202  ; D77 芯金前進ﾊｰﾌ
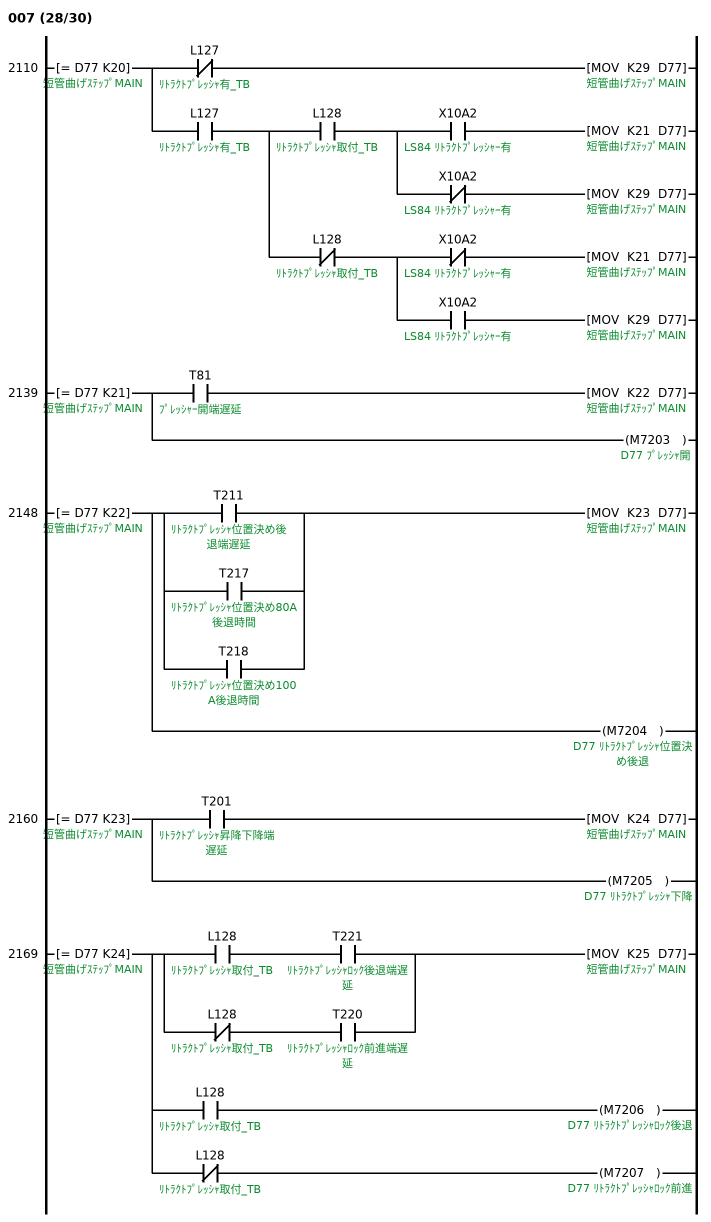
2110  LD=     D77 K20  ; 短管曲げｽﾃｯﾌﾟMAIN
      MPS
      ANI     L127  ; ﾘﾄﾗｸﾄﾌﾟﾚｯｼｬ有_TB
      MOV     K29 D77
      MPP
      AND     L127  ; ﾘﾄﾗｸﾄﾌﾟﾚｯｼｬ有_TB
      MPS
      AND     L128  ; ﾘﾄﾗｸﾄﾌﾟﾚｯｼｬ取付_TB
      MPS
      AND     X10A2  ; LS84 ﾘﾄﾗｸﾄﾌﾟﾚｯｼｬｰ有
      MOV     K21 D77
      MPP
      ANI     X10A2  ; LS84 ﾘﾄﾗｸﾄﾌﾟﾚｯｼｬｰ有
      MOV     K29 D77
      MPP
      ANI     L128  ; ﾘﾄﾗｸﾄﾌﾟﾚｯｼｬ取付_TB
      MPS
      ANI     X10A2  ; LS84 ﾘﾄﾗｸﾄﾌﾟﾚｯｼｬｰ有
      MOV     K21 D77
      MPP
      AND     X10A2  ; LS84 ﾘﾄﾗｸﾄﾌﾟﾚｯｼｬｰ有
      MOV     K29 D77
2139  LD=     D77 K21  ; 短管曲げｽﾃｯﾌﾟMAIN
      MPS
      AND     T81  ; ﾌﾟﾚｯｼｬｰ開端遅延
      MOV     K22 D77
      MPP
      OUT     M7203  ; D77 ﾌﾟﾚｯｼｬ開
2148  LD=     D77 K22  ; 短管曲げｽﾃｯﾌﾟMAIN
      MPS
      LD      T211  ; ﾘﾄﾗｸﾄﾌﾟﾚｯｼｬ位置決め後退端遅延
      OR      T217  ; ﾘﾄﾗｸﾄﾌﾟﾚｯｼｬ位置決め80A後退時間
      OR      T218  ; ﾘﾄﾗｸﾄﾌﾟﾚｯｼｬ位置決め100A後退時間
      ANB
      MOV     K23 D77
      MPP
      OUT     M7204  ; D77 ﾘﾄﾗｸﾄﾌﾟﾚｯｼｬ位置決め後退
2160  LD=     D77 K23  ; 短管曲げｽﾃｯﾌﾟMAIN
      MPS
      AND     T201  ; ﾘﾄﾗｸﾄﾌﾟﾚｯｼｬ昇降下降端遅延
      MOV     K24 D77
      MPP
      OUT     M7205  ; D77 ﾘﾄﾗｸﾄﾌﾟﾚｯｼｬ下降
2169  LD=     D77 K24  ; 短管曲げｽﾃｯﾌﾟMAIN
      MPS
      LD      L128  ; ﾘﾄﾗｸﾄﾌﾟﾚｯｼｬ取付_TB
      AND     T221  ; ﾘﾄﾗｸﾄﾌﾟﾚｯｼｬﾛｯｸ後退端遅延
      LDI     L128  ; ﾘﾄﾗｸﾄﾌﾟﾚｯｼｬ取付_TB
      AND     T220  ; ﾘﾄﾗｸﾄﾌﾟﾚｯｼｬﾛｯｸ前進端遅延
      ORB
      ANB
      MOV     K25 D77
      MRD
      AND     L128  ; ﾘﾄﾗｸﾄﾌﾟﾚｯｼｬ取付_TB
      OUT     M7206  ; D77 ﾘﾄﾗｸﾄﾌﾟﾚｯｼｬﾛｯｸ後退
      MPP
      ANI     L128  ; ﾘﾄﾗｸﾄﾌﾟﾚｯｼｬ取付_TB
      OUT     M7207  ; D77 ﾘﾄﾗｸﾄﾌﾟﾚｯｼｬﾛｯｸ前進
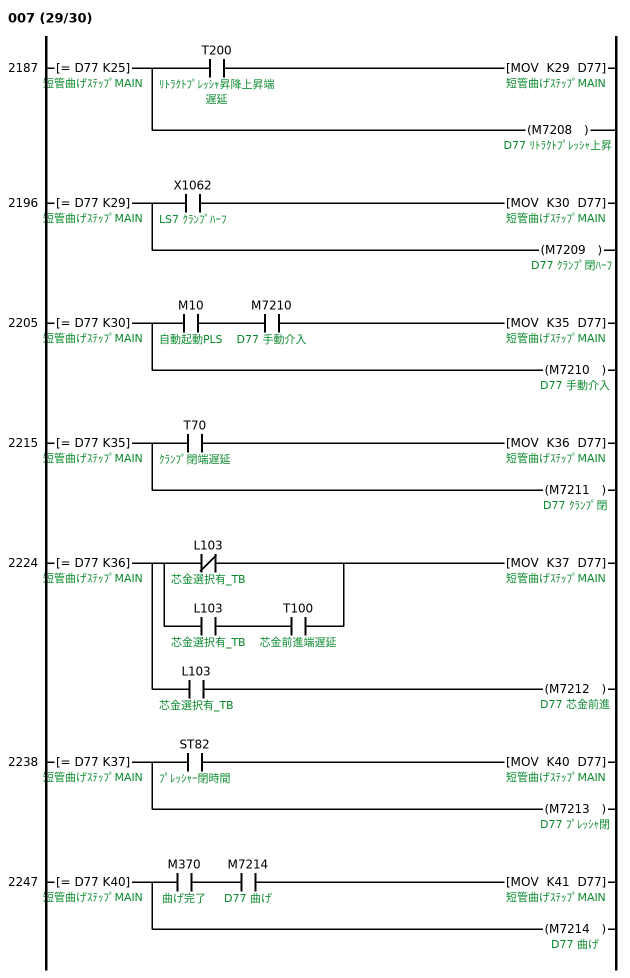
2187  LD=     D77 K25  ; 短管曲げｽﾃｯﾌﾟMAIN
      MPS
      AND     T200  ; ﾘﾄﾗｸﾄﾌﾟﾚｯｼｬ昇降上昇端遅延
      MOV     K29 D77
      MPP
      OUT     M7208  ; D77 ﾘﾄﾗｸﾄﾌﾟﾚｯｼｬ上昇
2196  LD=     D77 K29  ; 短管曲げｽﾃｯﾌﾟMAIN
      MPS
      AND     X1062  ; LS7 ｸﾗﾝﾌﾟﾊｰﾌ
      MOV     K30 D77
      MPP
      OUT     M7209  ; D77 ｸﾗﾝﾌﾟ閉ﾊｰﾌ
2205  LD=     D77 K30  ; 短管曲げｽﾃｯﾌﾟMAIN
      MPS
      AND     M10  ; 自動起動PLS
      AND     M7210  ; D77 手動介入
      MOV     K35 D77
      MPP
      OUT     M7210  ; D77 手動介入
2215  LD=     D77 K35  ; 短管曲げｽﾃｯﾌﾟMAIN
      MPS
      AND     T70  ; ｸﾗﾝﾌﾟ閉端遅延
      MOV     K36 D77
      MPP
      OUT     M7211  ; D77 ｸﾗﾝﾌﾟ閉
2224  LD=     D77 K36  ; 短管曲げｽﾃｯﾌﾟMAIN
      MPS
      LDI     L103  ; 芯金選択有_TB
      LD      L103  ; 芯金選択有_TB
      AND     T100  ; 芯金前進端遅延
      ORB
      ANB
      MOV     K37 D77
      MPP
      AND     L103  ; 芯金選択有_TB
      OUT     M7212  ; D77 芯金前進
2238  LD=     D77 K37  ; 短管曲げｽﾃｯﾌﾟMAIN
      MPS
      AND     ST82  ; ﾌﾟﾚｯｼｬｰ閉時間
      MOV     K40 D77
      MPP
      OUT     M7213  ; D77 ﾌﾟﾚｯｼｬ閉
2247  LD=     D77 K40  ; 短管曲げｽﾃｯﾌﾟMAIN
      MPS
      AND     M370  ; 曲げ完了
      AND     M7214  ; D77 曲げ
      MOV     K41 D77
      MPP
      OUT     M7214  ; D77 曲げ
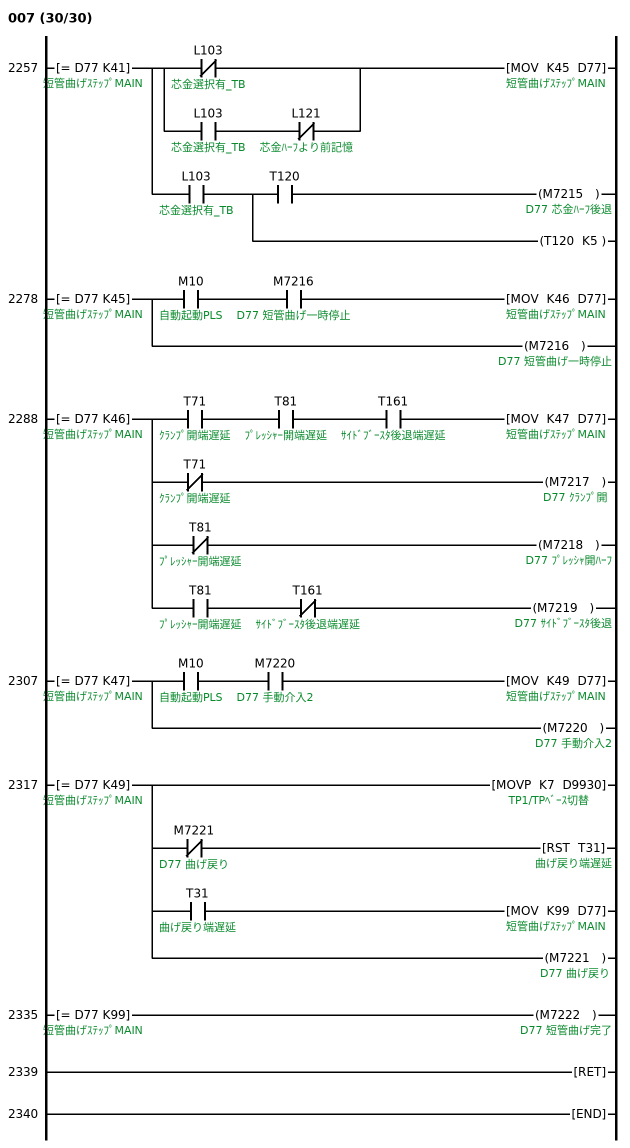
2257  LD=     D77 K41  ; 短管曲げｽﾃｯﾌﾟMAIN
      MPS
      LDI     L103  ; 芯金選択有_TB
      LD      L103  ; 芯金選択有_TB
      ANI     L121  ; 芯金ﾊｰﾌより前記憶
      ORB
      ANB
      MOV     K45 D77
      MPP
      AND     L103  ; 芯金選択有_TB
      MPS
      AND     T120
      OUT     M7215  ; D77 芯金ﾊｰﾌ後退
      MPP
      OUT     T120 K5
2278  LD=     D77 K45  ; 短管曲げｽﾃｯﾌﾟMAIN
      MPS
      AND     M10  ; 自動起動PLS
      AND     M7216  ; D77 短管曲げ一時停止
      MOV     K46 D77
      MPP
      OUT     M7216  ; D77 短管曲げ一時停止
2288  LD=     D77 K46  ; 短管曲げｽﾃｯﾌﾟMAIN
      MPS
      AND     T71  ; ｸﾗﾝﾌﾟ開端遅延
      AND     T81  ; ﾌﾟﾚｯｼｬｰ開端遅延
      AND     T161  ; ｻｲﾄﾞﾌﾞｰｽﾀ後退端遅延
      MOV     K47 D77
      MRD
      ANI     T71  ; ｸﾗﾝﾌﾟ開端遅延
      OUT     M7217  ; D77 ｸﾗﾝﾌﾟ開
      MRD
      ANI     T81  ; ﾌﾟﾚｯｼｬｰ開端遅延
      OUT     M7218  ; D77 ﾌﾟﾚｯｼｬ開ﾊｰﾌ
      MPP
      AND     T81  ; ﾌﾟﾚｯｼｬｰ開端遅延
      ANI     T161  ; ｻｲﾄﾞﾌﾞｰｽﾀ後退端遅延
      OUT     M7219  ; D77 ｻｲﾄﾞﾌﾞｰｽﾀ後退
2307  LD=     D77 K47  ; 短管曲げｽﾃｯﾌﾟMAIN
      MPS
      AND     M10  ; 自動起動PLS
      AND     M7220  ; D77 手動介入2
      MOV     K49 D77
      MPP
      OUT     M7220  ; D77 手動介入2
2317  LD=     D77 K49  ; 短管曲げｽﾃｯﾌﾟMAIN
      MOVP    K7 D9930
      MPS
      ANI     M7221  ; D77 曲げ戻り
      RST     T31  ; 曲げ戻り端遅延
      MRD
      AND     T31  ; 曲げ戻り端遅延
      MOV     K99 D77
      MPP
      OUT     M7221  ; D77 曲げ戻り
2335  LD=     D77 K99  ; 短管曲げｽﾃｯﾌﾟMAIN
      OUT     M7222  ; D77 短管曲げ完了
2339  RET
2340  END
END_PROGRAM

PROGRAM 008  // 自動準備
; 
      P800
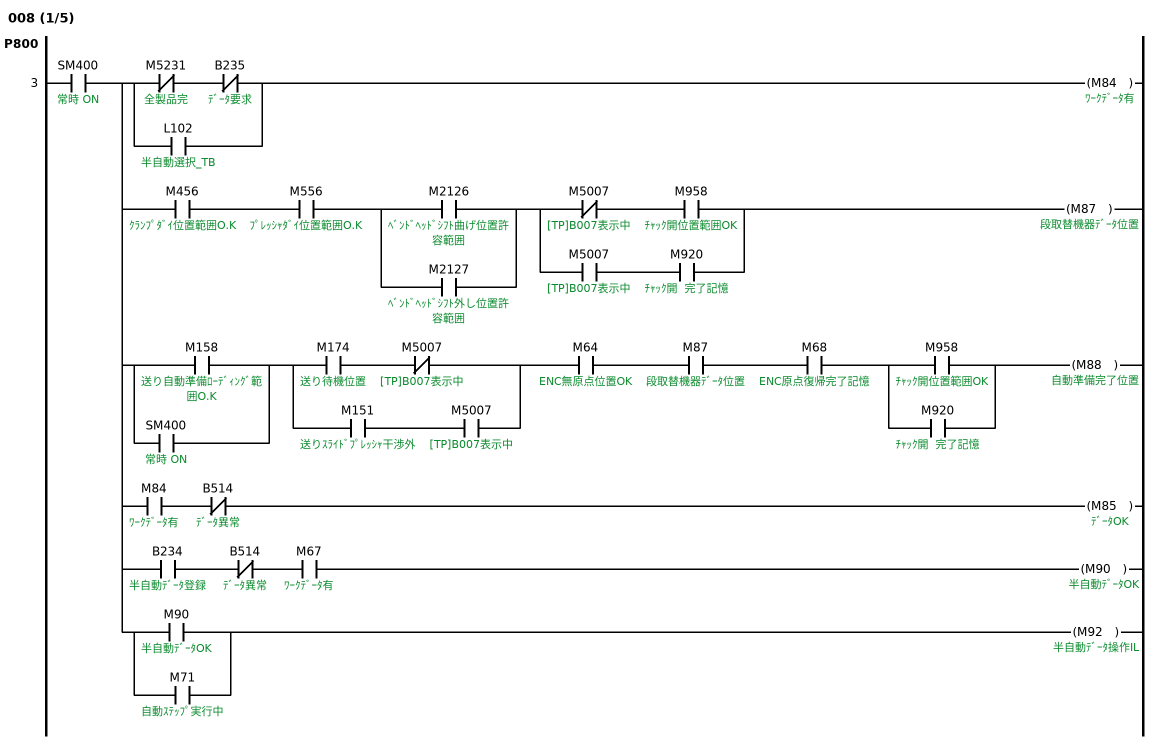
3     LD      SM400  ; 常時 ON
      MPS
      LDI     M5231  ; 全製品完
      ANI     B235  ; ﾃﾞｰﾀ要求
      OR      L102  ; 半自動選択_TB
      ANB
      OUT     M84  ; ﾜｰｸﾃﾞｰﾀ有
      MRD
      AND     M456  ; ｸﾗﾝﾌﾟﾀﾞｲ位置範囲O.K
      AND     M556  ; ﾌﾟﾚｯｼｬﾀﾞｲ位置範囲O.K
      LD      M2126  ; ﾍﾞﾝﾄﾞﾍｯﾄﾞｼﾌﾄ曲げ位置許容範囲
      OR      M2127  ; ﾍﾞﾝﾄﾞﾍｯﾄﾞｼﾌﾄ外し位置許容範囲
      ANB
      LDI     M5007  ; [TP]B007表示中
      AND     M958  ; ﾁｬｯｸ開位置範囲OK
      LD      M5007  ; [TP]B007表示中
      AND     M920  ; ﾁｬｯｸ開  完了記憶
      ORB
      ANB
      OUT     M87  ; 段取替機器ﾃﾞｰﾀ位置
      MRD
      LD      M158  ; 送り自動準備ﾛｰﾃﾞｨﾝｸﾞ範囲O.K
      OR      SM400  ; 常時 ON
      ANB
      LD      M174  ; 送り待機位置
      ANI     M5007  ; [TP]B007表示中
      LD      M151  ; 送りｽﾗｲﾄﾞﾌﾟﾚｯｼｬ干渉外
      AND     M5007  ; [TP]B007表示中
      ORB
      ANB
      AND     M64  ; ENC無原点位置OK
      AND     M87  ; 段取替機器ﾃﾞｰﾀ位置
      AND     M68  ; ENC原点復帰完了記憶
      LD      M958  ; ﾁｬｯｸ開位置範囲OK
      OR      M920  ; ﾁｬｯｸ開  完了記憶
      ANB
      OUT     M88  ; 自動準備完了位置
      MRD
      AND     M84  ; ﾜｰｸﾃﾞｰﾀ有
      ANI     B514  ; ﾃﾞｰﾀ異常
      OUT     M85  ; ﾃﾞｰﾀOK
      MRD
      AND     B234  ; 半自動ﾃﾞｰﾀ登録
      ANI     B514  ; ﾃﾞｰﾀ異常
      AND     M67  ; ﾜｰｸﾃﾞｰﾀ有
      OUT     M90  ; 半自動ﾃﾞｰﾀOK
      MPP
      LD      M90  ; 半自動ﾃﾞｰﾀOK
      OR      M71  ; 自動ｽﾃｯﾌﾟ実行中
      ANB
      OUT     M92  ; 半自動ﾃﾞｰﾀ操作IL
      P801
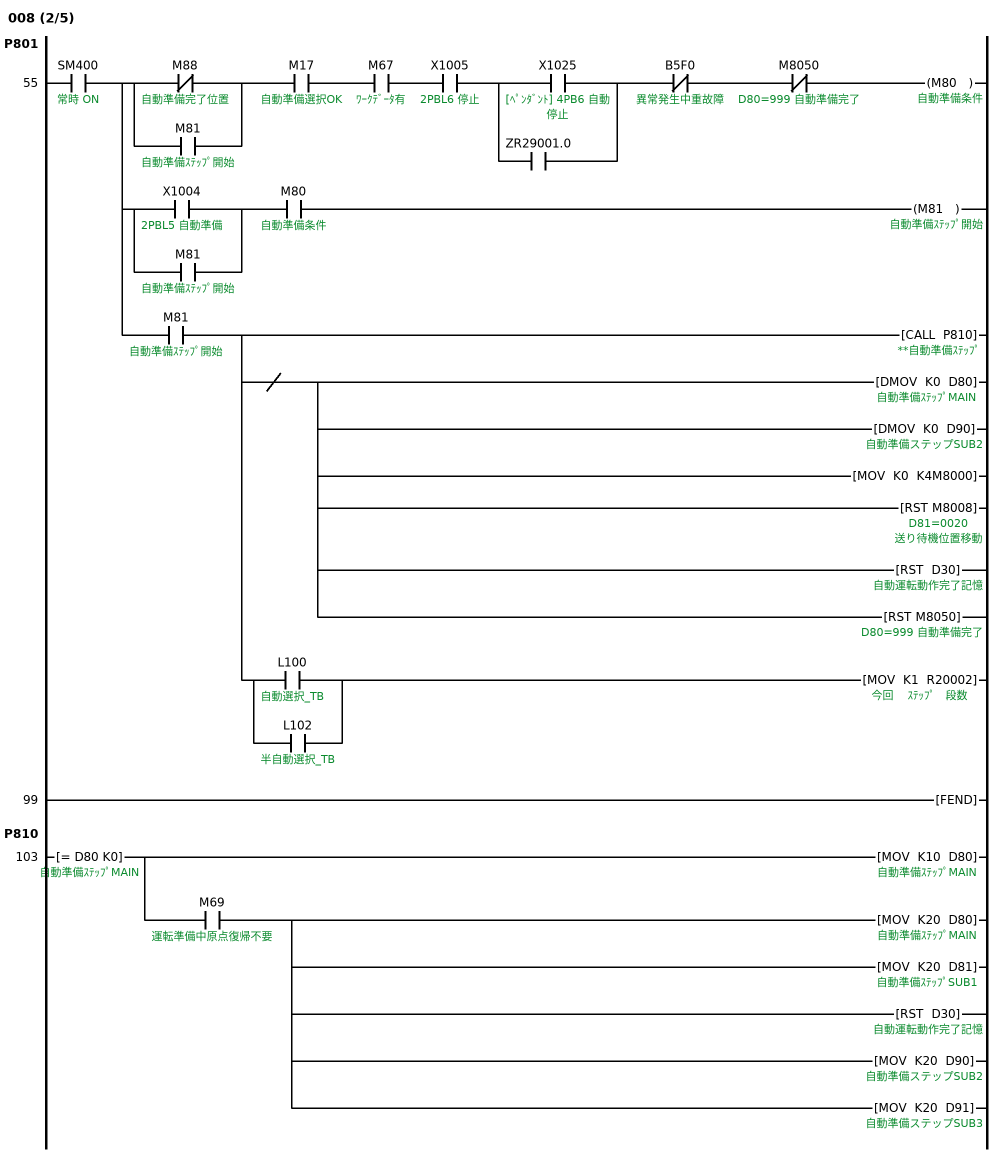
55    LD      SM400  ; 常時 ON
      MPS
      LDI     M88  ; 自動準備完了位置
      OR      M81  ; 自動準備ｽﾃｯﾌﾟ開始
      ANB
      AND     M17  ; 自動準備選択OK
      AND     M67  ; ﾜｰｸﾃﾞｰﾀ有
      AND     X1005  ; 2PBL6 停止
      LD      X1025  ; [ﾍﾟﾝﾀﾞﾝﾄ] 4PB6 自動 停止
      OR      ZR29001.0
      ANB
      ANI     B5F0  ; 異常発生中重故障
      ANI     M8050  ; D80=999 自動準備完了
      OUT     M80  ; 自動準備条件
      MRD
      LD      X1004  ; 2PBL5 自動準備
      OR      M81  ; 自動準備ｽﾃｯﾌﾟ開始
      ANB
      AND     M80  ; 自動準備条件
      OUT     M81  ; 自動準備ｽﾃｯﾌﾟ開始
      MPP
      AND     M81  ; 自動準備ｽﾃｯﾌﾟ開始
      CALL    P810  ; **自動準備ｽﾃｯﾌﾟ
      MPS
      INV
      DMOV    K0 D80  ; 自動準備ｽﾃｯﾌﾟMAIN
      DMOV    K0 D90  ; 自動準備ステップSUB2
      MOV     K0 K4M8000  ; D80=0010 原点復帰
      RST     M8008  ; D81=0020 送り待機位置移動
      RST     D30  ; 自動運転動作完了記憶
      RST     M8050  ; D80=999 自動準備完了
      MPP
      LD      L100  ; 自動選択_TB
      OR      L102  ; 半自動選択_TB
      ANB
      MOV     K1 R20002  ; 今回    ｽﾃｯﾌﾟ   段数
99    FEND
; 
      P810
103   LD=     D80 K0  ; 自動準備ｽﾃｯﾌﾟMAIN
      MOV     K10 D80
      AND     M69  ; 運転準備中原点復帰不要
      MOV     K20 D80
      MOV     K20 D81  ; 自動準備ｽﾃｯﾌﾟSUB1
      RST     D30  ; 自動運転動作完了記憶
      MOV     K20 D90
      MOV     K20 D91  ; 自動準備ステップSUB3
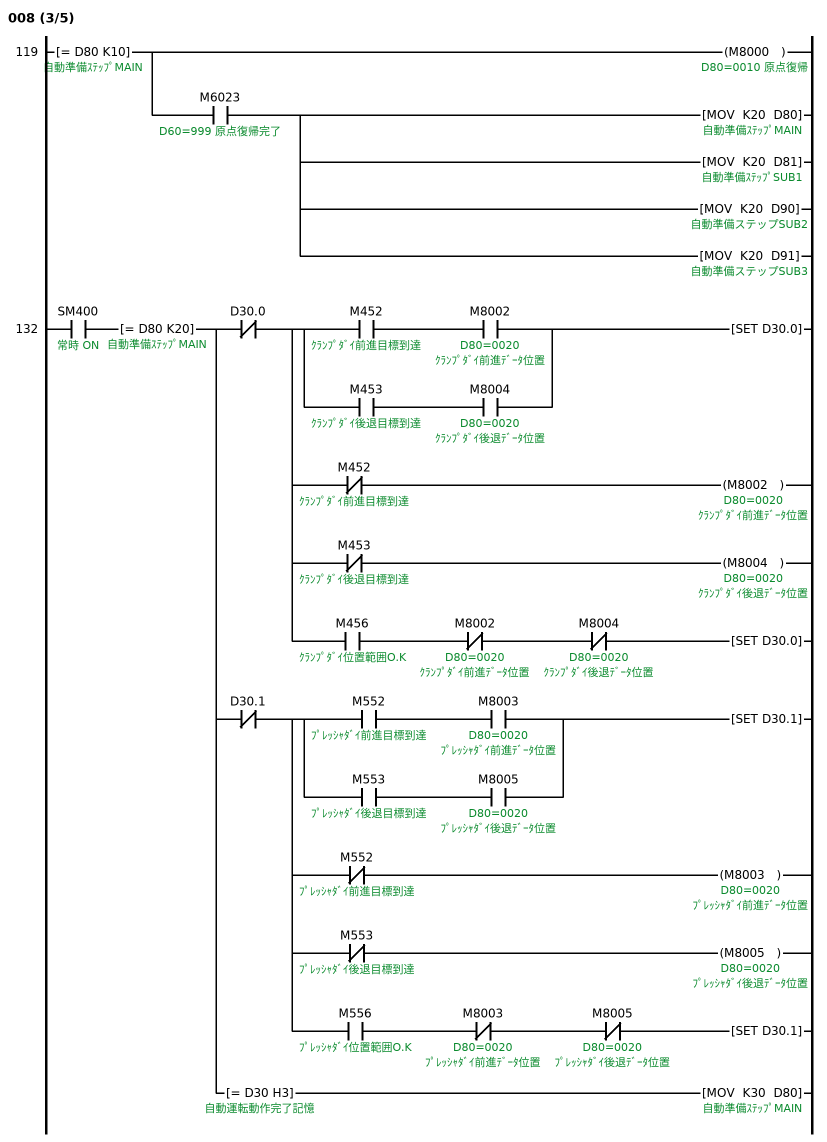
119   LD=     D80 K10  ; 自動準備ｽﾃｯﾌﾟMAIN
      OUT     M8000  ; D80=0010 原点復帰
      AND     M6023  ; D60=999 原点復帰完了
      MOV     K20 D80
      MOV     K20 D81
      MOV     K20 D90
      MOV     K20 D91
132   LD      SM400  ; 常時 ON
      AND=    D80 K20  ; 自動準備ｽﾃｯﾌﾟMAIN
      MPS
      ANI     D30.0
      MPS
      LD      M452  ; ｸﾗﾝﾌﾟﾀﾞｲ前進目標到達
      AND     M8002  ; D80=0020 ｸﾗﾝﾌﾟﾀﾞｲ前進ﾃﾞｰﾀ位置
      LD      M453  ; ｸﾗﾝﾌﾟﾀﾞｲ後退目標到達
      AND     M8004  ; D80=0020 ｸﾗﾝﾌﾟﾀﾞｲ後退ﾃﾞｰﾀ位置
      ORB
      ANB
      SET     D30.0
      MRD
      ANI     M452  ; ｸﾗﾝﾌﾟﾀﾞｲ前進目標到達
      OUT     M8002  ; D80=0020 ｸﾗﾝﾌﾟﾀﾞｲ前進ﾃﾞｰﾀ位置
      MRD
      ANI     M453  ; ｸﾗﾝﾌﾟﾀﾞｲ後退目標到達
      OUT     M8004  ; D80=0020 ｸﾗﾝﾌﾟﾀﾞｲ後退ﾃﾞｰﾀ位置
      MPP
      AND     M456  ; ｸﾗﾝﾌﾟﾀﾞｲ位置範囲O.K
      ANI     M8002  ; D80=0020 ｸﾗﾝﾌﾟﾀﾞｲ前進ﾃﾞｰﾀ位置
      ANI     M8004  ; D80=0020 ｸﾗﾝﾌﾟﾀﾞｲ後退ﾃﾞｰﾀ位置
      SET     D30.0
      MRD
      ANI     D30.1
      MPS
      LD      M552  ; ﾌﾟﾚｯｼｬﾀﾞｲ前進目標到達
      AND     M8003  ; D80=0020 ﾌﾟﾚｯｼｬﾀﾞｲ前進ﾃﾞｰﾀ位置
      LD      M553  ; ﾌﾟﾚｯｼｬﾀﾞｲ後退目標到達
      AND     M8005  ; D80=0020 ﾌﾟﾚｯｼｬﾀﾞｲ後退ﾃﾞｰﾀ位置
      ORB
      ANB
      SET     D30.1
      MRD
      ANI     M552  ; ﾌﾟﾚｯｼｬﾀﾞｲ前進目標到達
      OUT     M8003  ; D80=0020 ﾌﾟﾚｯｼｬﾀﾞｲ前進ﾃﾞｰﾀ位置
      MRD
      ANI     M553  ; ﾌﾟﾚｯｼｬﾀﾞｲ後退目標到達
      OUT     M8005  ; D80=0020 ﾌﾟﾚｯｼｬﾀﾞｲ後退ﾃﾞｰﾀ位置
      MPP
      AND     M556  ; ﾌﾟﾚｯｼｬﾀﾞｲ位置範囲O.K
      ANI     M8003  ; D80=0020 ﾌﾟﾚｯｼｬﾀﾞｲ前進ﾃﾞｰﾀ位置
      ANI     M8005  ; D80=0020 ﾌﾟﾚｯｼｬﾀﾞｲ後退ﾃﾞｰﾀ位置
      SET     D30.1
      MPP
      AND=    D30 H3  ; 自動運転動作完了記憶
      MOV     K30 D80
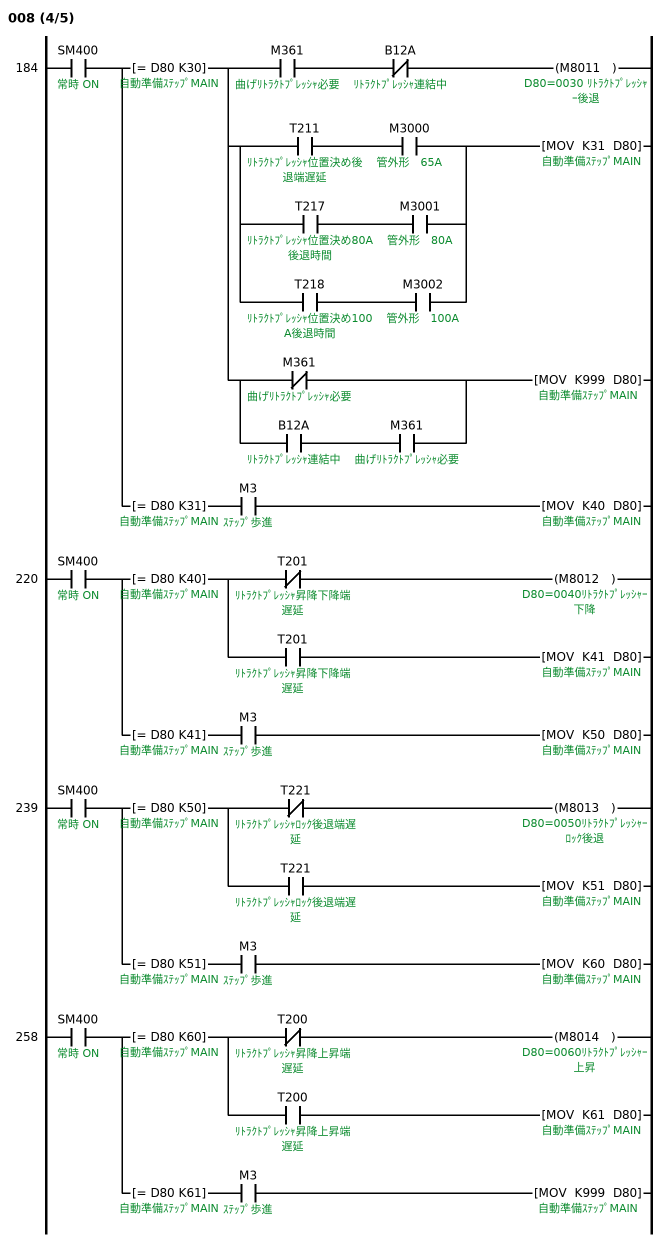
184   LD      SM400  ; 常時 ON
      MPS
      AND=    D80 K30  ; 自動準備ｽﾃｯﾌﾟMAIN
      MPS
      AND     M361  ; 曲げﾘﾄﾗｸﾄﾌﾟﾚｯｼｬ必要
      ANI     B12A  ; ﾘﾄﾗｸﾄﾌﾟﾚｯｼｬ連結中
      OUT     M8011  ; D80=0030 ﾘﾄﾗｸﾄﾌﾟﾚｯｼｬｰ後退
      MRD
      LD      T211  ; ﾘﾄﾗｸﾄﾌﾟﾚｯｼｬ位置決め後退端遅延
      AND     M3000  ; 管外形　65A
      LD      T217  ; ﾘﾄﾗｸﾄﾌﾟﾚｯｼｬ位置決め80A後退時間
      AND     M3001  ; 管外形　80A
      ORB
      LD      T218  ; ﾘﾄﾗｸﾄﾌﾟﾚｯｼｬ位置決め100A後退時間
      AND     M3002  ; 管外形　100A
      ORB
      ANB
      MOV     K31 D80
      MPP
      LDI     M361  ; 曲げﾘﾄﾗｸﾄﾌﾟﾚｯｼｬ必要
      LD      B12A  ; ﾘﾄﾗｸﾄﾌﾟﾚｯｼｬ連結中
      AND     M361  ; 曲げﾘﾄﾗｸﾄﾌﾟﾚｯｼｬ必要
      ORB
      ANB
      MOV     K999 D80
      MPP
      AND=    D80 K31  ; 自動準備ｽﾃｯﾌﾟMAIN
      AND     M3  ; ｽﾃｯﾌﾟ歩進
      MOV     K40 D80
220   LD      SM400  ; 常時 ON
      MPS
      AND=    D80 K40  ; 自動準備ｽﾃｯﾌﾟMAIN
      MPS
      ANI     T201  ; ﾘﾄﾗｸﾄﾌﾟﾚｯｼｬ昇降下降端遅延
      OUT     M8012  ; D80=0040ﾘﾄﾗｸﾄﾌﾟﾚｯｼｬｰ下降
      MPP
      AND     T201  ; ﾘﾄﾗｸﾄﾌﾟﾚｯｼｬ昇降下降端遅延
      MOV     K41 D80
      MPP
      AND=    D80 K41  ; 自動準備ｽﾃｯﾌﾟMAIN
      AND     M3  ; ｽﾃｯﾌﾟ歩進
      MOV     K50 D80
239   LD      SM400  ; 常時 ON
      MPS
      AND=    D80 K50  ; 自動準備ｽﾃｯﾌﾟMAIN
      MPS
      ANI     T221  ; ﾘﾄﾗｸﾄﾌﾟﾚｯｼｬﾛｯｸ後退端遅延
      OUT     M8013  ; D80=0050ﾘﾄﾗｸﾄﾌﾟﾚｯｼｬｰﾛｯｸ後退
      MPP
      AND     T221  ; ﾘﾄﾗｸﾄﾌﾟﾚｯｼｬﾛｯｸ後退端遅延
      MOV     K51 D80
      MPP
      AND=    D80 K51  ; 自動準備ｽﾃｯﾌﾟMAIN
      AND     M3  ; ｽﾃｯﾌﾟ歩進
      MOV     K60 D80
258   LD      SM400  ; 常時 ON
      MPS
      AND=    D80 K60  ; 自動準備ｽﾃｯﾌﾟMAIN
      MPS
      ANI     T200  ; ﾘﾄﾗｸﾄﾌﾟﾚｯｼｬ昇降上昇端遅延
      OUT     M8014  ; D80=0060ﾘﾄﾗｸﾄﾌﾟﾚｯｼｬｰ上昇
      MPP
      AND     T200  ; ﾘﾄﾗｸﾄﾌﾟﾚｯｼｬ昇降上昇端遅延
      MOV     K61 D80
      MPP
      AND=    D80 K61  ; 自動準備ｽﾃｯﾌﾟMAIN
      AND     M3  ; ｽﾃｯﾌﾟ歩進
      MOV     K999 D80
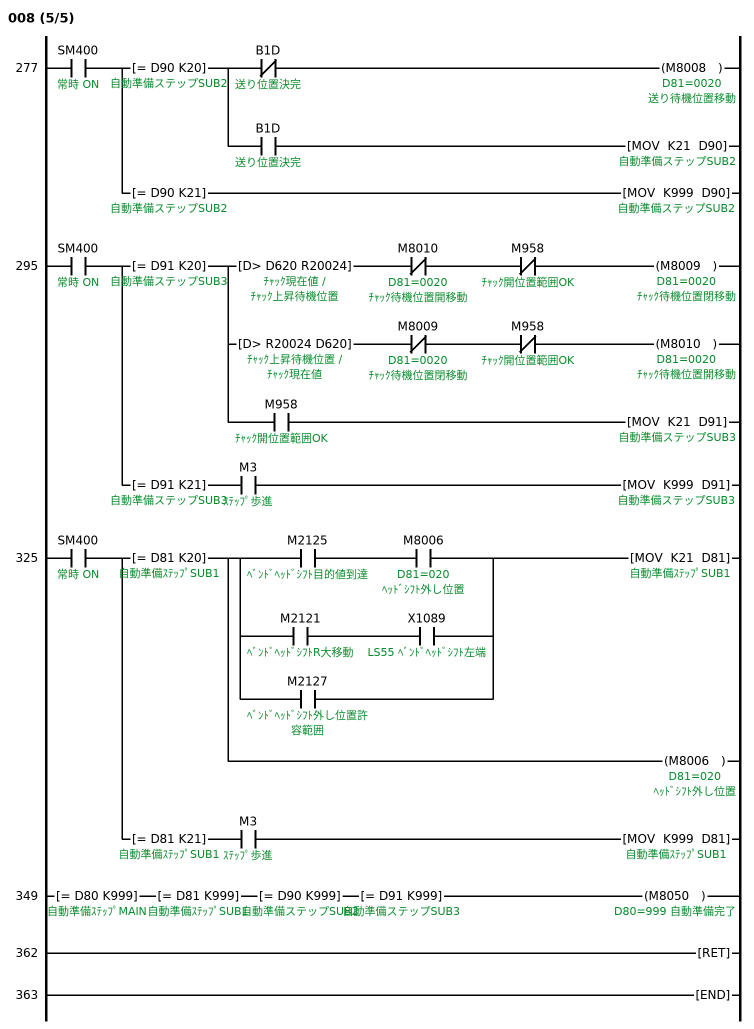
277   LD      SM400  ; 常時 ON
      MPS
      AND=    D90 K20  ; 自動準備ステップSUB2
      MPS
      ANI     B1D  ; 送り位置決完
      OUT     M8008  ; D81=0020 送り待機位置移動
      MPP
      AND     B1D  ; 送り位置決完
      MOV     K21 D90
      MPP
      AND=    D90 K21  ; 自動準備ステップSUB2
      MOV     K999 D90
295   LD      SM400  ; 常時 ON
      MPS
      AND=    D91 K20  ; 自動準備ステップSUB3
      MPS
      ANDD>   D620 R20024  ; ﾁｬｯｸ現在値 / ﾁｬｯｸ上昇待機位置
      ANI     M8010  ; D81=0020 ﾁｬｯｸ待機位置開移動
      ANI     M958  ; ﾁｬｯｸ開位置範囲OK
      OUT     M8009  ; D81=0020 ﾁｬｯｸ待機位置閉移動
      MRD
      ANDD>   R20024 D620  ; ﾁｬｯｸ上昇待機位置 / ﾁｬｯｸ現在値
      ANI     M8009  ; D81=0020 ﾁｬｯｸ待機位置閉移動
      ANI     M958  ; ﾁｬｯｸ開位置範囲OK
      OUT     M8010  ; D81=0020 ﾁｬｯｸ待機位置開移動
      MPP
      AND     M958  ; ﾁｬｯｸ開位置範囲OK
      MOV     K21 D91
      MPP
      AND=    D91 K21  ; 自動準備ステップSUB3
      AND     M3  ; ｽﾃｯﾌﾟ歩進
      MOV     K999 D91
325   LD      SM400  ; 常時 ON
      MPS
      AND=    D81 K20  ; 自動準備ｽﾃｯﾌﾟSUB1
      MPS
      LD      M2125  ; ﾍﾞﾝﾄﾞﾍｯﾄﾞｼﾌﾄ目的値到達
      AND     M8006  ; D81=020 ﾍｯﾄﾞｼﾌﾄ外し位置
      LD      M2121  ; ﾍﾞﾝﾄﾞﾍｯﾄﾞｼﾌﾄR大移動
      AND     X1089  ; LS55 ﾍﾞﾝﾄﾞﾍｯﾄﾞｼﾌﾄ左端
      ORB
      OR      M2127  ; ﾍﾞﾝﾄﾞﾍｯﾄﾞｼﾌﾄ外し位置許容範囲
      ANB
      MOV     K21 D81
      MPP
      OUT     M8006  ; D81=020 ﾍｯﾄﾞｼﾌﾄ外し位置
      MPP
      AND=    D81 K21  ; 自動準備ｽﾃｯﾌﾟSUB1
      AND     M3  ; ｽﾃｯﾌﾟ歩進
      MOV     K999 D81
349   LD=     D80 K999  ; 自動準備ｽﾃｯﾌﾟMAIN
      AND=    D81 K999  ; 自動準備ｽﾃｯﾌﾟSUB1
      AND=    D90 K999  ; 自動準備ステップSUB2
      AND=    D91 K999  ; 自動準備ステップSUB3
      OUT     M8050  ; D80=999 自動準備完了
362   RET
363   END
END_PROGRAM

PROGRAM 010  // 手動SV
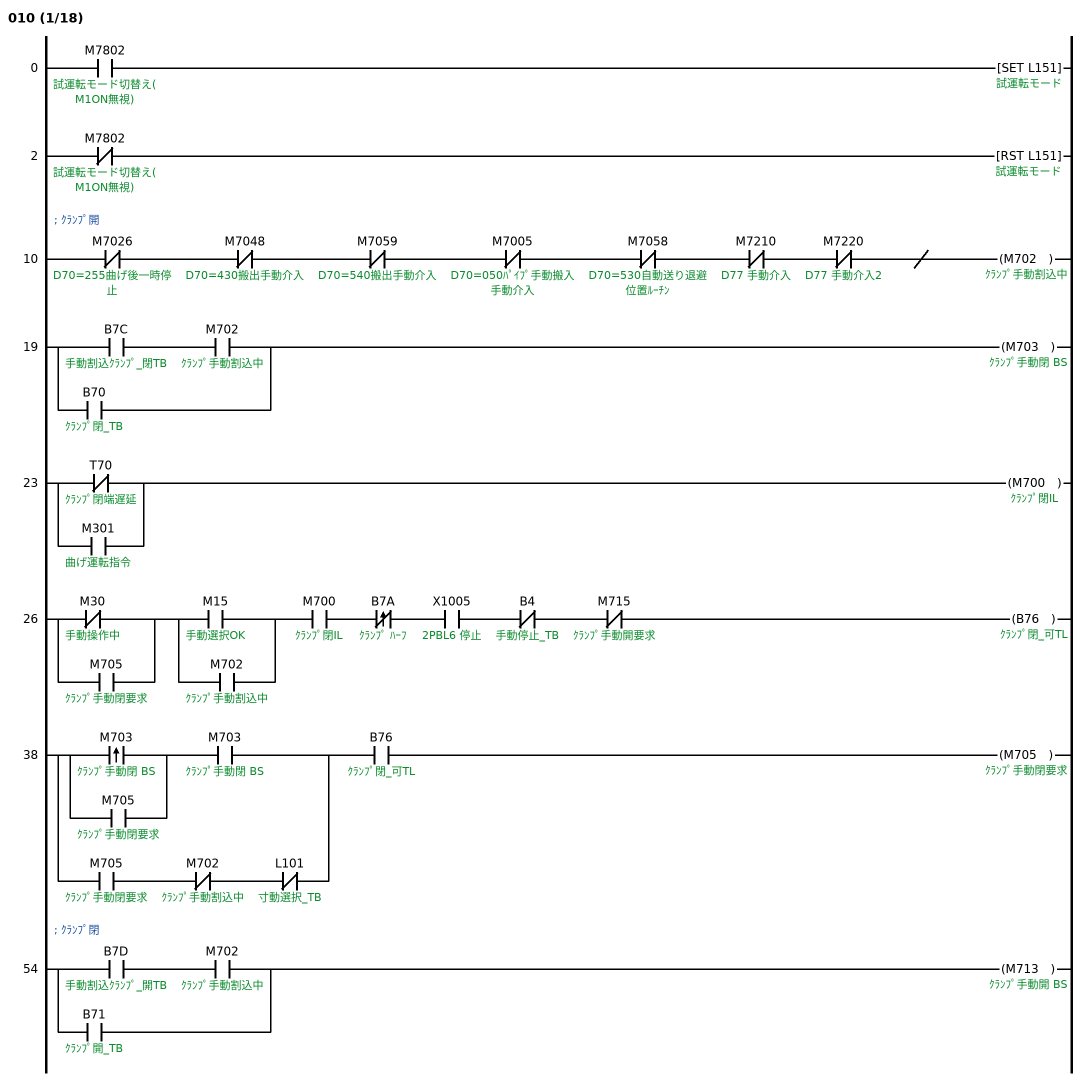
0     LD      M7802  ; 試運転モード切替え(M1ON無視)
      SET     L151  ; 試運転モード
2     LDI     M7802  ; 試運転モード切替え(M1ON無視)
      RST     L151  ; 試運転モード
; ｸﾗﾝﾌﾟ開
10    LDI     M7026  ; D70=255曲げ後一時停止
      ANI     M7048  ; D70=430搬出手動介入
      ANI     M7059  ; D70=540搬出手動介入
      ANI     M7005  ; D70=050ﾊﾟｲﾌﾟ手動搬入手動介入
      ANI     M7058  ; D70=530自動送り退避位置ﾙｰﾁﾝ
      ANI     M7210  ; D77 手動介入
      ANI     M7220  ; D77 手動介入2
      INV
      OUT     M702  ; ｸﾗﾝﾌﾟ手動割込中
19    LD      B7C  ; 手動割込ｸﾗﾝﾌﾟ_閉TB
      AND     M702  ; ｸﾗﾝﾌﾟ手動割込中
      OR      B70  ; ｸﾗﾝﾌﾟ閉_TB
      OUT     M703  ; ｸﾗﾝﾌﾟ手動閉 BS
23    LDI     T70  ; ｸﾗﾝﾌﾟ閉端遅延
      OR      M301  ; 曲げ運転指令
      OUT     M700  ; ｸﾗﾝﾌﾟ閉IL
26    LDI     M30  ; 手動操作中
      OR      M705  ; ｸﾗﾝﾌﾟ手動閉要求
      LD      M15  ; 手動選択OK
      OR      M702  ; ｸﾗﾝﾌﾟ手動割込中
      ANB
      AND     M700  ; ｸﾗﾝﾌﾟ閉IL
      ANDPI   B7A  ; ｸﾗﾝﾌﾟ ﾊｰﾌ
      AND     X1005  ; 2PBL6 停止
      ANI     B4  ; 手動停止_TB
      ANI     M715  ; ｸﾗﾝﾌﾟ手動開要求
      OUT     B76  ; ｸﾗﾝﾌﾟ閉_可TL
38    LDP     M703  ; ｸﾗﾝﾌﾟ手動閉 BS
      OR      M705  ; ｸﾗﾝﾌﾟ手動閉要求
      AND     M703  ; ｸﾗﾝﾌﾟ手動閉 BS
      LD      M705  ; ｸﾗﾝﾌﾟ手動閉要求
      ANI     M702  ; ｸﾗﾝﾌﾟ手動割込中
      ANI     L101  ; 寸動選択_TB
      ORB
      AND     B76  ; ｸﾗﾝﾌﾟ閉_可TL
      OUT     M705  ; ｸﾗﾝﾌﾟ手動閉要求
; ｸﾗﾝﾌﾟ閉
54    LD      B7D  ; 手動割込ｸﾗﾝﾌﾟ_開TB
      AND     M702  ; ｸﾗﾝﾌﾟ手動割込中
      OR      B71  ; ｸﾗﾝﾌﾟ開_TB
      OUT     M713  ; ｸﾗﾝﾌﾟ手動開 BS
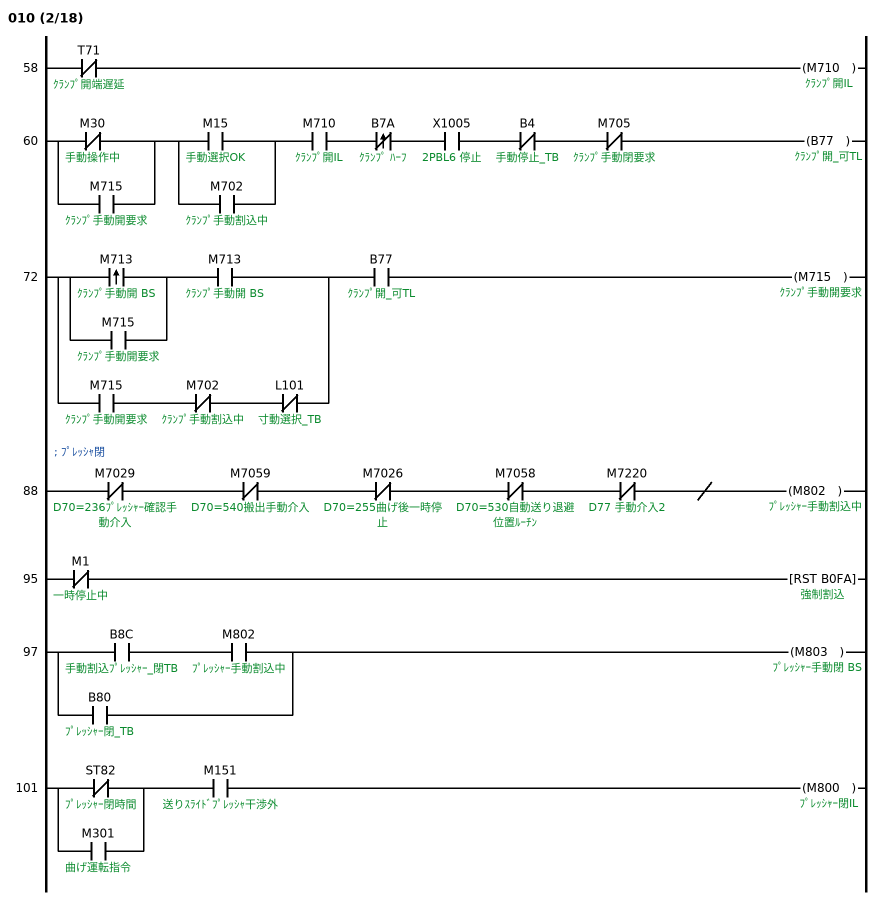
58    LDI     T71  ; ｸﾗﾝﾌﾟ開端遅延
      OUT     M710  ; ｸﾗﾝﾌﾟ開IL
60    LDI     M30  ; 手動操作中
      OR      M715  ; ｸﾗﾝﾌﾟ手動開要求
      LD      M15  ; 手動選択OK
      OR      M702  ; ｸﾗﾝﾌﾟ手動割込中
      ANB
      AND     M710  ; ｸﾗﾝﾌﾟ開IL
      ANDPI   B7A  ; ｸﾗﾝﾌﾟ ﾊｰﾌ
      AND     X1005  ; 2PBL6 停止
      ANI     B4  ; 手動停止_TB
      ANI     M705  ; ｸﾗﾝﾌﾟ手動閉要求
      OUT     B77  ; ｸﾗﾝﾌﾟ開_可TL
72    LDP     M713  ; ｸﾗﾝﾌﾟ手動開 BS
      OR      M715  ; ｸﾗﾝﾌﾟ手動開要求
      AND     M713  ; ｸﾗﾝﾌﾟ手動開 BS
      LD      M715  ; ｸﾗﾝﾌﾟ手動開要求
      ANI     M702  ; ｸﾗﾝﾌﾟ手動割込中
      ANI     L101  ; 寸動選択_TB
      ORB
      AND     B77  ; ｸﾗﾝﾌﾟ開_可TL
      OUT     M715  ; ｸﾗﾝﾌﾟ手動開要求
; ﾌﾟﾚｯｼｬ閉
88    LDI     M7029  ; D70=236ﾌﾟﾚｯｼｬｰ確認手動介入
      ANI     M7059  ; D70=540搬出手動介入
      ANI     M7026  ; D70=255曲げ後一時停止
      ANI     M7058  ; D70=530自動送り退避位置ﾙｰﾁﾝ
      ANI     M7220  ; D77 手動介入2
      INV
      OUT     M802  ; ﾌﾟﾚｯｼｬｰ手動割込中
95    LDI     M1  ; 一時停止中
      RST     B0FA  ; 強制割込
97    LD      B8C  ; 手動割込ﾌﾟﾚｯｼｬｰ_閉TB
      AND     M802  ; ﾌﾟﾚｯｼｬｰ手動割込中
      OR      B80  ; ﾌﾟﾚｯｼｬｰ閉_TB
      OUT     M803  ; ﾌﾟﾚｯｼｬｰ手動閉 BS
101   LDI     ST82  ; ﾌﾟﾚｯｼｬｰ閉時間
      OR      M301  ; 曲げ運転指令
      AND     M151  ; 送りｽﾗｲﾄﾞﾌﾟﾚｯｼｬ干渉外
      OUT     M800  ; ﾌﾟﾚｯｼｬｰ閉IL
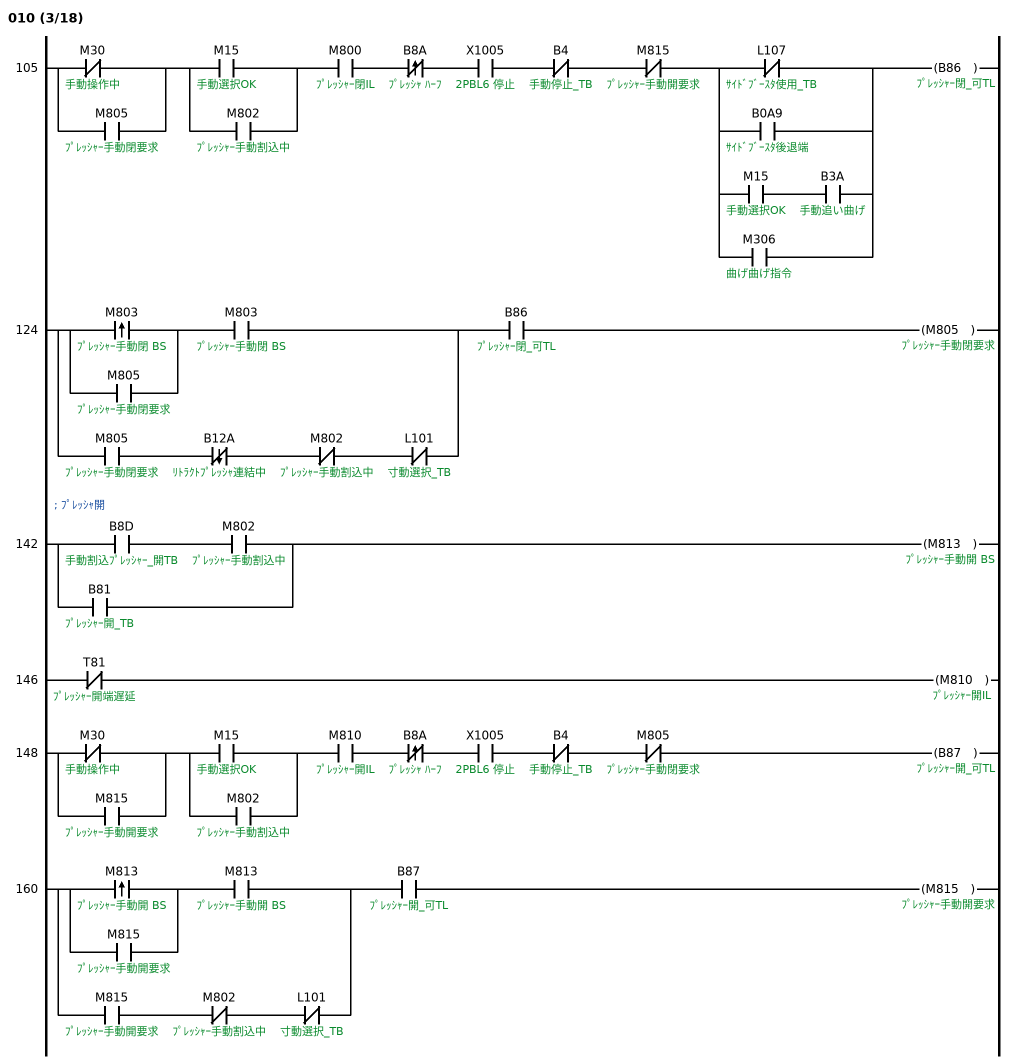
105   LDI     M30  ; 手動操作中
      OR      M805  ; ﾌﾟﾚｯｼｬｰ手動閉要求
      LD      M15  ; 手動選択OK
      OR      M802  ; ﾌﾟﾚｯｼｬｰ手動割込中
      ANB
      AND     M800  ; ﾌﾟﾚｯｼｬｰ閉IL
      ANDPI   B8A  ; ﾌﾟﾚｯｼｬ ﾊｰﾌ
      AND     X1005  ; 2PBL6 停止
      ANI     B4  ; 手動停止_TB
      ANI     M815  ; ﾌﾟﾚｯｼｬｰ手動開要求
      LDI     L107  ; ｻｲﾄﾞﾌﾞｰｽﾀ使用_TB
      OR      B0A9  ; ｻｲﾄﾞﾌﾞｰｽﾀ後退端
      LD      M15  ; 手動選択OK
      AND     B3A  ; 手動追い曲げ
      ORB
      OR      M306  ; 曲げ曲げ指令
      ANB
      OUT     B86  ; ﾌﾟﾚｯｼｬｰ閉_可TL
124   LDP     M803  ; ﾌﾟﾚｯｼｬｰ手動閉 BS
      OR      M805  ; ﾌﾟﾚｯｼｬｰ手動閉要求
      AND     M803  ; ﾌﾟﾚｯｼｬｰ手動閉 BS
      LD      M805  ; ﾌﾟﾚｯｼｬｰ手動閉要求
      ANDFI   B12A  ; ﾘﾄﾗｸﾄﾌﾟﾚｯｼｬ連結中
      ANI     M802  ; ﾌﾟﾚｯｼｬｰ手動割込中
      ANI     L101  ; 寸動選択_TB
      ORB
      AND     B86  ; ﾌﾟﾚｯｼｬｰ閉_可TL
      OUT     M805  ; ﾌﾟﾚｯｼｬｰ手動閉要求
; ﾌﾟﾚｯｼｬ開
142   LD      B8D  ; 手動割込ﾌﾟﾚｯｼｬｰ_開TB
      AND     M802  ; ﾌﾟﾚｯｼｬｰ手動割込中
      OR      B81  ; ﾌﾟﾚｯｼｬｰ開_TB
      OUT     M813  ; ﾌﾟﾚｯｼｬｰ手動開 BS
146   LDI     T81  ; ﾌﾟﾚｯｼｬｰ開端遅延
      OUT     M810  ; ﾌﾟﾚｯｼｬｰ開IL
148   LDI     M30  ; 手動操作中
      OR      M815  ; ﾌﾟﾚｯｼｬｰ手動開要求
      LD      M15  ; 手動選択OK
      OR      M802  ; ﾌﾟﾚｯｼｬｰ手動割込中
      ANB
      AND     M810  ; ﾌﾟﾚｯｼｬｰ開IL
      ANDPI   B8A  ; ﾌﾟﾚｯｼｬ ﾊｰﾌ
      AND     X1005  ; 2PBL6 停止
      ANI     B4  ; 手動停止_TB
      ANI     M805  ; ﾌﾟﾚｯｼｬｰ手動閉要求
      OUT     B87  ; ﾌﾟﾚｯｼｬｰ開_可TL
160   LDP     M813  ; ﾌﾟﾚｯｼｬｰ手動開 BS
      OR      M815  ; ﾌﾟﾚｯｼｬｰ手動開要求
      AND     M813  ; ﾌﾟﾚｯｼｬｰ手動開 BS
      LD      M815  ; ﾌﾟﾚｯｼｬｰ手動開要求
      ANI     M802  ; ﾌﾟﾚｯｼｬｰ手動割込中
      ANI     L101  ; 寸動選択_TB
      ORB
      AND     B87  ; ﾌﾟﾚｯｼｬｰ開_可TL
      OUT     M815  ; ﾌﾟﾚｯｼｬｰ手動開要求
